LIN {X 0.002,Y -498.772,Z 962.107,A 0.000,B 0.000,C 90.000,E1 235.229} C_DIS
LIN {X -0.113,Y -494.068,Z 962.095,A 0.000,B 0.000,C 90.000,E1 233.130} C_DIS
LIN {X -0.156,Y -489.223,Z 962.083,A 0.000,B 0.000,C 90.000,E1 231.009} C_DIS
LIN {X -0.020,Y -484.237,Z 962.071,A 0.000,B 0.000,C 90.000,E1 228.852} C_DIS
LIN {X -0.074,Y -479.355,Z 962.059,A 0.000,B 0.000,C 90.000,E1 226.701} C_DIS
LIN {X -0.051,Y -475.254,Z 962.049,A 0.000,B 0.000,C 90.000,E1 224.838} C_DIS
LIN {X 0.307,Y -470.435,Z 962.037,A 0.000,B 0.000,C 90.000,E1 222.609} C_DIS
LIN {X -0.169,Y -466.298,Z 962.026,A 0.000,B 0.000,C 90.000,E1 220.782} C_DIS
LIN {X 0.117,Y -463.523,Z 962.019,A 0.000,B 0.000,C 90.000,E1 219.483} C_DIS
LIN {X -0.073,Y -458.612,Z 962.007,A 0.000,B 0.000,C 90.000,E1 217.282} C_DIS
LIN {X -0.034,Y -454.314,Z 961.996,A 0.000,B 0.000,C 90.000,E1 215.358} C_DIS
LIN {X 0.095,Y -449.373,Z 961.984,A 0.000,B 0.000,C 90.000,E1 213.086} C_DIS
LIN {X 0.228,Y -444.453,Z 961.971,A 0.000,B 0.000,C 90.000,E1 210.797} C_DIS
LIN {X -0.008,Y -439.493,Z 961.959,A 0.000,B 0.000,C 90.000,E1 208.537} C_DIS
LIN {X -0.041,Y -435.155,Z 961.948,A 0.000,B 0.000,C 90.000,E1 206.565} C_DIS
LIN {X 0.022,Y -431.464,Z 961.938,A 0.000,B 0.000,C 90.000,E1 204.899} C_DIS
LIN {X 0.016,Y -428.364,Z 961.931,A 0.000,B 0.000,C 90.000,E1 203.567} C_DIS
LIN {X -0.074,Y -421.639,Z 961.914,A 0.000,B 0.000,C 90.000,E1 200.556} C_DIS
LIN {X -0.162,Y -418.818,Z 961.907,A 0.000,B 0.000,C 90.000,E1 199.214} C_DIS
LIN {X 0.032,Y -414.002,Z 961.893,A 0.000,B 0.000,C 90.000,E1 196.804} C_DIS
LIN {X 0.082,Y -411.371,Z 961.886,A 0.000,B 0.000,C 90.000,E1 195.426} C_DIS
LIN {X -0.005,Y -407.947,Z 961.876,A 0.000,B 0.000,C 90.000,E1 193.716} C_DIS
LIN {X -0.164,Y -405.246,Z 961.869,A 0.000,B 0.000,C 90.000,E1 192.355} C_DIS
LIN {X -0.068,Y -401.253,Z 961.857,A 0.000,B 0.000,C 90.000,E1 190.254} C_DIS
LIN {X -0.122,Y -397.922,Z 961.847,A 0.000,B 0.000,C 90.000,E1 188.511} C_DIS
LIN {X -0.111,Y -392.119,Z 961.830,A 0.000,B 0.000,C 90.000,E1 185.334} C_DIS
LIN {X -0.093,Y -389.441,Z 961.820,A 0.000,B 0.000,C 90.000,E1 183.555} C_DIS
LIN {X -0.182,Y -388.975,Z 961.818,A 0.000,B 0.000,C 90.000,E1 183.212} C_DIS
LIN {X -0.048,Y -388.111,Z 961.812,A 0.000,B 0.000,C 90.000,E1 182.121} C_DIS
LIN {X 0.165,Y -387.977,Z 961.808,A 0.000,B 0.000,C 90.000,E1 181.375} C_DIS
LIN {X -0.023,Y -388.436,Z 961.804,A 0.000,B 0.000,C 90.000,E1 180.688} C_DIS
LIN {X -0.115,Y -388.908,Z 961.802,A 0.000,B 0.000,C 90.000,E1 180.344} C_DIS
LIN {X 0.138,Y -390.130,Z 961.799,A 0.000,B 0.000,C 90.000,E1 179.771} C_DIS
LIN {X 0.191,Y -391.585,Z 961.797,A 0.000,B 0.000,C 90.000,E1 179.370} C_DIS
LIN {X 0.109,Y -393.003,Z 961.795,A 0.000,B 0.000,C 90.000,E1 179.026} C_DIS
LIN {X 0.031,Y -394.990,Z 961.793,A 0.000,B 0.000,C 90.000,E1 178.682} C_DIS
LIN {X 0.104,Y -398.169,Z 961.790,A 0.000,B 0.000,C 90.000,E1 178.224} C_DIS
LIN {X -0.090,Y -402.312,Z 961.788,A 0.000,B 0.000,C 90.000,E1 177.764} C_DIS
LIN {X -0.070,Y -408.333,Z 961.784,A 0.000,B 0.000,C 90.000,E1 177.192} C_DIS
LIN {X -0.198,Y -420.662,Z 961.778,A 0.000,B 0.000,C 90.000,E1 176.102} C_DIS
LIN {X -0.071,Y -429.525,Z 961.774,A 0.000,B 0.000,C 90.000,E1 175.298} C_DIS
LIN {X -0.092,Y -438.634,Z 961.769,A 0.000,B 0.000,C 90.000,E1 174.489} C_DIS
LIN {X 0.100,Y -447.490,Z 961.765,A 0.000,B 0.000,C 90.000,E1 173.628} C_DIS
LIN {X -0.043,Y -454.687,Z 961.761,A 0.000,B 0.000,C 90.000,E1 172.932} C_DIS
LIN {X -0.092,Y -460.322,Z 961.758,A 0.000,B 0.000,C 90.000,E1 172.356} C_DIS
LIN {X 0.185,Y -468.563,Z 961.753,A 0.000,B 0.000,C 90.000,E1 171.432} C_DIS
LIN {X 0.154,Y -474.872,Z 961.749,A 0.000,B 0.000,C 90.000,E1 170.735} C_DIS
LIN {X 0.189,Y -482.568,Z 961.744,A 0.000,B 0.000,C 90.000,E1 169.803} C_DIS
LIN {X 0.051,Y -488.804,Z 961.739,A 0.000,B 0.000,C 90.000,E1 169.050} C_DIS
LIN {X 0.203,Y -495.887,Z 961.734,A 0.000,B 0.000,C 90.000,E1 168.117} C_DIS
LIN {X 0.132,Y -500.316,Z 961.731,A 0.000,B 0.000,C 90.000,E1 167.521} C_DIS
LIN {X -0.132,Y -508.811,Z 961.724,A 0.000,B 0.000,C 90.000,E1 166.353} C_DIS
LIN {X -0.165,Y -516.756,Z 961.718,A 0.000,B 0.000,C 90.000,E1 165.172} C_DIS
LIN {X -0.265,Y -523.259,Z 961.712,A 0.000,B 0.000,C 90.000,E1 164.157} C_DIS
LIN {X 0.228,Y -529.654,Z 961.706,A 0.000,B 0.000,C 90.000,E1 163.087} C_DIS
LIN {X -0.270,Y -540.981,Z 961.696,A 0.000,B 0.000,C 90.000,E1 161.275} C_DIS
LIN {X -0.336,Y -548.482,Z 961.689,A 0.000,B 0.000,C 90.000,E1 160.007} C_DIS
LIN {X 0.063,Y -552.643,Z 961.685,A 0.000,B 0.000,C 90.000,E1 159.263} C_DIS
LIN {X 0.083,Y -558.360,Z 961.679,A 0.000,B 0.000,C 90.000,E1 158.284} C_DIS
LIN {X 0.171,Y -561.441,Z 961.676,A 0.000,B 0.000,C 90.000,E1 157.720} C_DIS
LIN {X 0.199,Y -567.306,Z 961.670,A 0.000,B 0.000,C 90.000,E1 156.613} C_DIS
LIN {X 0.094,Y -572.082,Z 961.665,A 0.000,B 0.000,C 90.000,E1 155.665} C_DIS
LIN {X 0.207,Y -575.439,Z 961.661,A 0.000,B 0.000,C 90.000,E1 154.973} C_DIS
LIN {X -0.175,Y -578.579,Z 961.657,A 0.000,B 0.000,C 90.000,E1 154.332} C_DIS
LIN {X 0.174,Y -584.416,Z 961.650,A 0.000,B 0.000,C 90.000,E1 152.948} C_DIS
LIN {X 0.072,Y -587.609,Z 961.645,A 0.000,B 0.000,C 90.000,E1 152.153} C_DIS
LIN {X -0.203,Y -592.331,Z 961.638,A 0.000,B 0.000,C 90.000,E1 150.845} C_DIS
LIN {X 0.207,Y -595.985,Z 961.632,A 0.000,B 0.000,C 90.000,E1 149.744} C_DIS
LIN {X -0.231,Y -601.336,Z 961.623,A 0.000,B 0.000,C 90.000,E1 148.201} C_DIS
LIN {X -0.051,Y -608.089,Z 961.612,A 0.000,B 0.000,C 90.000,E1 146.087} C_DIS
LIN {X -0.141,Y -614.086,Z 961.602,A 0.000,B 0.000,C 90.000,E1 144.276} C_DIS
LIN {X -0.226,Y -619.902,Z 961.591,A 0.000,B 0.000,C 90.000,E1 142.477} C_DIS
LIN {X 0.032,Y -624.035,Z 961.584,A 0.000,B 0.000,C 90.000,E1 141.170} C_DIS
LIN {X 0.312,Y -631.372,Z 961.572,A 0.000,B 0.000,C 90.000,E1 138.852} C_DIS
LIN {X -0.048,Y -638.178,Z 961.560,A 0.000,B 0.000,C 90.000,E1 136.863} C_DIS
LIN {X 0.258,Y -644.183,Z 961.551,A 0.000,B 0.000,C 90.000,E1 135.081} C_DIS
LIN {X 0.159,Y -652.114,Z 961.538,A 0.000,B 0.000,C 90.000,E1 132.852} C_DIS
LIN {X 0.330,Y -660.280,Z 961.526,A 0.000,B 0.000,C 90.000,E1 130.620} C_DIS
LIN {X -0.148,Y -664.928,Z 961.519,A 0.000,B 0.000,C 90.000,E1 129.439} C_DIS
LIN {X -0.106,Y -667.632,Z 961.515,A 0.000,B 0.000,C 90.000,E1 128.705} C_DIS
LIN {X -0.048,Y -671.179,Z 961.510,A 0.000,B 0.000,C 90.000,E1 127.729} C_DIS
LIN {X 0.168,Y -675.377,Z 961.503,A 0.000,B 0.000,C 90.000,E1 126.503} C_DIS
LIN {X -0.098,Y -677.796,Z 961.499,A 0.000,B 0.000,C 90.000,E1 125.804} C_DIS
LIN {X -0.174,Y -681.560,Z 961.492,A 0.000,B 0.000,C 90.000,E1 124.612} C_DIS
LIN {X 0.184,Y -684.351,Z 961.487,A 0.000,B 0.000,C 90.000,E1 123.627} C_DIS
LIN {X -0.177,Y -687.537,Z 961.480,A 0.000,B 0.000,C 90.000,E1 122.467} C_DIS
LIN {X -0.126,Y -689.987,Z 961.475,A 0.000,B 0.000,C 90.000,E1 121.514} C_DIS
LIN {X 0.190,Y -692.197,Z 961.470,A 0.000,B 0.000,C 90.000,E1 120.541} C_DIS
LIN {X -0.292,Y -693.641,Z 961.466,A 0.000,B 0.000,C 90.000,E1 119.873} C_DIS
LIN {X -0.161,Y -694.952,Z 961.462,A 0.000,B 0.000,C 90.000,E1 119.155} C_DIS
LIN {X -0.115,Y -696.465,Z 961.455,A 0.000,B 0.000,C 90.000,E1 117.975} C_DIS
LIN {X 0.043,Y -697.251,Z 961.451,A 0.000,B 0.000,C 90.000,E1 117.257} C_DIS
LIN {X -0.206,Y -698.130,Z 961.445,A 0.000,B 0.000,C 90.000,E1 116.104} C_DIS
LIN {X 0.187,Y -698.621,Z 961.438,A 0.000,B 0.000,C 90.000,E1 114.899} C_DIS
LIN {X -0.210,Y -698.721,Z 961.436,A 0.000,B 0.000,C 90.000,E1 114.463} C_DIS
LIN {X 0.054,Y -698.680,Z 961.435,A 0.000,B 0.000,C 90.000,E1 114.207} C_DIS
LIN {X -0.340,Y -698.341,Z 961.432,A 0.000,B 0.000,C 90.000,E1 113.770} C_DIS
LIN {X 0.182,Y -697.167,Z 961.429,A 0.000,B 0.000,C 90.000,E1 113.259} C_DIS
LIN {X 0.165,Y -696.462,Z 961.428,A 0.000,B 0.000,C 90.000,E1 113.025} C_DIS
LIN {X -0.220,Y -695.014,Z 961.427,A 0.000,B 0.000,C 90.000,E1 112.823} C_DIS
LIN {X -0.117,Y -692.305,Z 961.425,A 0.000,B 0.000,C 90.000,E1 112.461} C_DIS
LIN {X 0.004,Y -691.173,Z 961.424,A 0.000,B 0.000,C 90.000,E1 112.333} C_DIS
LIN {X 0.121,Y -689.434,Z 961.423,A 0.000,B 0.000,C 90.000,E1 112.206} C_DIS
LIN {X -0.041,Y -683.525,Z 961.422,A 0.000,B 0.000,C 90.000,E1 111.950} C_DIS
LIN {X 0.173,Y -679.388,Z 961.421,A 0.000,B 0.000,C 90.000,E1 111.791} C_DIS
LIN {X -0.228,Y -677.435,Z 961.421,A 0.000,B 0.000,C 90.000,E1 111.770} C_DIS
LIN {X -0.251,Y -674.935,Z 961.421,A 0.000,B 0.000,C 90.000,E1 111.716} C_DIS
LIN {X -0.095,Y -667.646,Z 961.420,A 0.000,B 0.000,C 90.000,E1 111.663} C_DIS
LIN {X -0.128,Y -628.953,Z 961.420,A 0.000,B 0.000,C 90.000,E1 111.663} C_DIS
LIN {X 0.227,Y -623.063,Z 961.420,A 0.000,B 0.000,C 90.000,E1 111.535} C_DIS
LIN {X -0.156,Y -616.228,Z 961.419,A 0.000,B 0.000,C 90.000,E1 111.408} C_DIS
LIN {X 0.114,Y -609.362,Z 961.418,A 0.000,B 0.000,C 90.000,E1 111.153} C_DIS
LIN {X 0.021,Y -606.468,Z 961.417,A 0.000,B 0.000,C 90.000,E1 111.046} C_DIS
LIN {X -0.108,Y -599.985,Z 961.415,A 0.000,B 0.000,C 90.000,E1 110.737} C_DIS
LIN {X 0.314,Y -593.503,Z 961.413,A 0.000,B 0.000,C 90.000,E1 110.301} C_DIS
LIN {X 0.129,Y -584.030,Z 961.409,A 0.000,B 0.000,C 90.000,E1 109.631} C_DIS
LIN {X 0.293,Y -575.275,Z 961.406,A 0.000,B 0.000,C 90.000,E1 108.960} C_DIS
LIN {X -0.143,Y -567.394,Z 961.403,A 0.000,B 0.000,C 90.000,E1 108.544} C_DIS
LIN {X 0.139,Y -553.077,Z 961.399,A 0.000,B 0.000,C 90.000,E1 107.819} C_DIS
LIN {X -0.272,Y -550.970,Z 961.398,A 0.000,B 0.000,C 90.000,E1 107.638} C_DIS
LIN {X 0.213,Y -550.938,Z 961.398,A 0.000,B 0.000,C 90.000,E1 107.583} C_DIS
LIN {X -0.167,Y -550.493,Z 961.397,A 0.000,B 0.000,C 90.000,E1 107.457} C_DIS
LIN {X 0.192,Y -550.350,Z 961.394,A 0.000,B 0.000,C 90.000,E1 106.858} C_DIS
LIN {X 0.057,Y -550.977,Z 961.384,A 0.000,B 0.000,C 90.000,E1 105.190} C_DIS
LIN {X 0.153,Y -552.146,Z 961.372,A 0.000,B 0.000,C 90.000,E1 102.939} C_DIS
LIN {X -0.246,Y -554.640,Z 961.355,A 0.000,B 0.000,C 90.000,E1 99.905} C_DIS
LIN {X -0.245,Y -555.958,Z 961.347,A 0.000,B 0.000,C 90.000,E1 98.511} C_DIS
LIN {X 0.251,Y -557.272,Z 961.339,A 0.000,B 0.000,C 90.000,E1 97.068} C_DIS
LIN {X 0.149,Y -558.100,Z 961.333,A 0.000,B 0.000,C 90.000,E1 95.967} C_DIS
LIN {X 0.066,Y -559.114,Z 961.326,A 0.000,B 0.000,C 90.000,E1 94.588} C_DIS
LIN {X 0.175,Y -560.219,Z 961.315,A 0.000,B 0.000,C 90.000,E1 92.636} C_DIS
LIN {X 0.096,Y -560.910,Z 961.307,A 0.000,B 0.000,C 90.000,E1 91.260} C_DIS
LIN {X -0.080,Y -561.411,Z 961.301,A 0.000,B 0.000,C 90.000,E1 90.172} C_DIS
LIN {X -0.150,Y -561.855,Z 961.293,A 0.000,B 0.000,C 90.000,E1 88.797} C_DIS
LIN {X -0.104,Y -562.253,Z 961.284,A 0.000,B 0.000,C 90.000,E1 87.135} C_DIS
LIN {X -0.113,Y -562.489,Z 961.276,A 0.000,B 0.000,C 90.000,E1 85.755} C_DIS
LIN {X -0.026,Y -562.713,Z 961.267,A 0.000,B 0.000,C 90.000,E1 84.090} C_DIS
LIN {X 0.031,Y -562.924,Z 961.260,A 0.000,B 0.000,C 90.000,E1 82.704} C_DIS
LIN {X 0.245,Y -563.276,Z 961.250,A 0.000,B 0.000,C 90.000,E1 81.027} C_DIS
LIN {X -0.226,Y -564.154,Z 961.238,A 0.000,B 0.000,C 90.000,E1 78.870} C_DIS
LIN {X -0.171,Y -565.125,Z 961.227,A 0.000,B 0.000,C 90.000,E1 76.937} C_DIS
LIN {X -0.134,Y -566.143,Z 961.218,A 0.000,B 0.000,C 90.000,E1 75.283} C_DIS
LIN {X 0.239,Y -567.482,Z 961.208,A 0.000,B 0.000,C 90.000,E1 73.323} C_DIS
LIN {X -0.238,Y -568.369,Z 961.200,A 0.000,B 0.000,C 90.000,E1 72.000} C_DIS
LIN {X 0.172,Y -569.291,Z 961.191,A 0.000,B 0.000,C 90.000,E1 70.315} C_DIS
LIN {X -0.284,Y -570.013,Z 961.182,A 0.000,B 0.000,C 90.000,E1 68.720} C_DIS
LIN {X 0.236,Y -570.324,Z 961.177,A 0.000,B 0.000,C 90.000,E1 67.847} C_DIS
LIN {X 0.023,Y -570.847,Z 961.168,A 0.000,B 0.000,C 90.000,E1 66.230} C_DIS
LIN {X 0.219,Y -571.193,Z 961.160,A 0.000,B 0.000,C 90.000,E1 64.845} C_DIS
LIN {X -0.265,Y -571.517,Z 961.151,A 0.000,B 0.000,C 90.000,E1 63.256} C_DIS
LIN {X 0.182,Y -571.720,Z 961.144,A 0.000,B 0.000,C 90.000,E1 61.847} C_DIS
LIN {X -0.100,Y -571.827,Z 961.136,A 0.000,B 0.000,C 90.000,E1 60.511} C_DIS
LIN {X 0.080,Y -572.018,Z 961.126,A 0.000,B 0.000,C 90.000,E1 58.584} C_DIS
LIN {X -0.188,Y -572.093,Z 961.118,A 0.000,B 0.000,C 90.000,E1 57.248} C_DIS
LIN {X -0.020,Y -571.806,Z 961.109,A 0.000,B 0.000,C 90.000,E1 55.595} C_DIS
LIN {X 0.329,Y -571.460,Z 961.101,A 0.000,B 0.000,C 90.000,E1 54.196} C_DIS
LIN {X 0.073,Y -570.984,Z 961.095,A 0.000,B 0.000,C 90.000,E1 53.130} C_DIS
LIN {X 0.156,Y -570.251,Z 961.089,A 0.000,B 0.000,C 90.000,E1 52.029} C_DIS
LIN {X -0.125,Y -569.304,Z 961.083,A 0.000,B 0.000,C 90.000,E1 50.964} C_DIS
LIN {X 0.294,Y -568.235,Z 961.077,A 0.000,B 0.000,C 90.000,E1 49.828} C_DIS
LIN {X 0.215,Y -567.228,Z 961.072,A 0.000,B 0.000,C 90.000,E1 49.013} C_DIS
LIN {X -0.303,Y -566.025,Z 961.068,A 0.000,B 0.000,C 90.000,E1 48.243} C_DIS
LIN {X 0.064,Y -564.090,Z 961.062,A 0.000,B 0.000,C 90.000,E1 47.106} C_DIS
LIN {X 0.372,Y -561.923,Z 961.056,A 0.000,B 0.000,C 90.000,E1 45.972} C_DIS
LIN {X 0.189,Y -559.978,Z 961.051,A 0.000,B 0.000,C 90.000,E1 45.162} C_DIS
LIN {X -0.012,Y -557.802,Z 961.046,A 0.000,B 0.000,C 90.000,E1 44.352} C_DIS
LIN {X -0.236,Y -555.254,Z 961.042,A 0.000,B 0.000,C 90.000,E1 43.542} C_DIS
LIN {X 0.264,Y -553.483,Z 961.039,A 0.000,B 0.000,C 90.000,E1 42.933} C_DIS
LIN {X -0.028,Y -551.510,Z 961.036,A 0.000,B 0.000,C 90.000,E1 42.405} C_DIS
LIN {X 0.086,Y -548.196,Z 961.031,A 0.000,B 0.000,C 90.000,E1 41.553} C_DIS
LIN {X -0.037,Y -545.280,Z 961.027,A 0.000,B 0.000,C 90.000,E1 40.862} C_DIS
LIN {X -0.029,Y -542.661,Z 961.024,A 0.000,B 0.000,C 90.000,E1 40.297} C_DIS
LIN {X 0.021,Y -539.856,Z 961.021,A 0.000,B 0.000,C 90.000,E1 39.725} C_DIS
LIN {X -0.013,Y -533.798,Z 961.014,A 0.000,B 0.000,C 90.000,E1 38.588} C_DIS
LIN {X -0.035,Y -528.791,Z 961.010,A 0.000,B 0.000,C 90.000,E1 37.729} C_DIS
LIN {X 0.032,Y -522.690,Z 961.004,A 0.000,B 0.000,C 90.000,E1 36.710} C_DIS
LIN {X -0.234,Y -518.057,Z 961.000,A 0.000,B 0.000,C 90.000,E1 36.011} C_DIS
LIN {X -0.004,Y -512.279,Z 960.995,A 0.000,B 0.000,C 90.000,E1 35.105} C_DIS
LIN {X -0.166,Y -508.091,Z 960.992,A 0.000,B 0.000,C 90.000,E1 34.532} C_DIS
LIN {X 0.057,Y -503.632,Z 960.988,A 0.000,B 0.000,C 90.000,E1 33.913} C_DIS
LIN {X 0.244,Y -498.877,Z 960.985,A 0.000,B 0.000,C 90.000,E1 33.293} C_DIS
LIN {X -0.086,Y -495.051,Z 960.983,A 0.000,B 0.000,C 90.000,E1 32.880} C_DIS
LIN {X 0.081,Y -488.398,Z 960.979,A 0.000,B 0.000,C 90.000,E1 32.133} C_DIS
LIN {X 0.073,Y -481.531,Z 960.975,A 0.000,B 0.000,C 90.000,E1 31.416} C_DIS
LIN {X -0.107,Y -471.350,Z 960.969,A 0.000,B 0.000,C 90.000,E1 30.463} C_DIS
LIN {X 0.183,Y -463.949,Z 960.965,A 0.000,B 0.000,C 90.000,E1 29.745} C_DIS
LIN {X 0.171,Y -455.058,Z 960.961,A 0.000,B 0.000,C 90.000,E1 28.949} C_DIS
LIN {X 0.248,Y -442.802,Z 960.955,A 0.000,B 0.000,C 90.000,E1 27.897} C_DIS
LIN {X -0.116,Y -423.164,Z 960.946,A 0.000,B 0.000,C 90.000,E1 26.232} C_DIS
LIN {X 0.066,Y -406.759,Z 960.937,A 0.000,B 0.000,C 90.000,E1 24.643} C_DIS
LIN {X 0.050,Y -398.631,Z 960.932,A 0.000,B 0.000,C 90.000,E1 23.770} C_DIS
LIN {X 0.158,Y -393.390,Z 960.928,A 0.000,B 0.000,C 90.000,E1 23.078} C_DIS
LIN {X 0.117,Y -391.309,Z 960.926,A 0.000,B 0.000,C 90.000,E1 22.642} C_DIS
LIN {X 0.065,Y -390.232,Z 960.923,A 0.000,B 0.000,C 90.000,E1 22.206} C_DIS
LIN {X 0.084,Y -389.878,Z 960.922,A 0.000,B 0.000,C 90.000,E1 22.025} C_DIS
LIN {X 0.049,Y -389.531,Z 960.919,A 0.000,B 0.000,C 90.000,E1 21.408} C_DIS
LIN {X -0.156,Y -389.967,Z 960.913,A 0.000,B 0.000,C 90.000,E1 20.301} C_DIS
LIN {X 0.152,Y -392.234,Z 960.899,A 0.000,B 0.000,C 90.000,E1 17.764} C_DIS
LIN {X -0.017,Y -395.491,Z 960.883,A 0.000,B 0.000,C 90.000,E1 14.954} C_DIS
LIN {X 0.092,Y -399.231,Z 960.867,A 0.000,B 0.000,C 90.000,E1 12.119} C_DIS
LIN {X 0.072,Y -403.658,Z 960.852,A 0.000,B 0.000,C 90.000,E1 9.321} C_DIS
LIN {X 0.020,Y -408.661,Z 960.836,A 0.000,B 0.000,C 90.000,E1 6.549} C_DIS
LIN {X 0.118,Y -415.635,Z 960.817,A 0.000,B 0.000,C 90.000,E1 3.094} C_DIS
LIN {X -0.144,Y -420.986,Z 960.804,A 0.000,B 0.000,C 90.000,E1 0.745} C_DIS
LIN {X 0.000,Y -422.737,Z 960.800,A 0.000,B 0.000,C 90.000,E1 360.000} C_DIS
LIN {X -0.053,Y -425.183,Z 960.796,A 0.000,B 0.000,C 90.000,E1 359.312} C_DIS
LIN {X -0.118,Y -428.115,Z 960.793,A 0.000,B 0.000,C 90.000,E1 358.797} C_DIS
LIN {X 0.142,Y -429.485,Z 960.792,A 0.000,B 0.000,C 90.000,E1 358.511} C_DIS
LIN {X -0.025,Y -432.070,Z 960.790,A 0.000,B 0.000,C 90.000,E1 358.282} C_DIS
LIN {X 0.079,Y -434.973,Z 960.789,A 0.000,B 0.000,C 90.000,E1 357.993} C_DIS
LIN {X -0.159,Y -441.329,Z 960.787,A 0.000,B 0.000,C 90.000,E1 357.650} C_DIS
LIN {X -0.090,Y -450.033,Z 960.784,A 0.000,B 0.000,C 90.000,E1 357.192} C_DIS
LIN {X -0.185,Y -465.315,Z 960.780,A 0.000,B 0.000,C 90.000,E1 356.388} C_DIS
LIN {X -0.060,Y -473.709,Z 960.777,A 0.000,B 0.000,C 90.000,E1 355.927} C_DIS
LIN {X 0.093,Y -483.670,Z 960.774,A 0.000,B 0.000,C 90.000,E1 355.355} C_DIS
LIN {X -0.153,Y -493.694,Z 960.771,A 0.000,B 0.000,C 90.000,E1 354.837} C_DIS
LIN {X -0.022,Y -503.392,Z 960.768,A 0.000,B 0.000,C 90.000,E1 354.261} C_DIS
LIN {X -0.111,Y -512.933,Z 960.765,A 0.000,B 0.000,C 90.000,E1 353.685} C_DIS
LIN {X 0.191,Y -523.897,Z 960.761,A 0.000,B 0.000,C 90.000,E1 352.932} C_DIS
LIN {X -0.019,Y -531.408,Z 960.758,A 0.000,B 0.000,C 90.000,E1 352.413} C_DIS
LIN {X 0.158,Y -539.663,Z 960.754,A 0.000,B 0.000,C 90.000,E1 351.724} C_DIS
LIN {X -0.121,Y -546.547,Z 960.751,A 0.000,B 0.000,C 90.000,E1 351.141} C_DIS
LIN {X 0.086,Y -550.532,Z 960.749,A 0.000,B 0.000,C 90.000,E1 350.735} C_DIS
LIN {X 0.116,Y -556.731,Z 960.745,A 0.000,B 0.000,C 90.000,E1 350.095} C_DIS
LIN {X 0.204,Y -562.520,Z 960.741,A 0.000,B 0.000,C 90.000,E1 349.398} C_DIS
LIN {X -0.033,Y -566.889,Z 960.738,A 0.000,B 0.000,C 90.000,E1 348.870} C_DIS
LIN {X -0.051,Y -572.834,Z 960.734,A 0.000,B 0.000,C 90.000,E1 348.049} C_DIS
LIN {X -0.007,Y -578.239,Z 960.729,A 0.000,B 0.000,C 90.000,E1 347.229} C_DIS
LIN {X -0.243,Y -584.758,Z 960.723,A 0.000,B 0.000,C 90.000,E1 346.172} C_DIS
LIN {X 0.319,Y -590.677,Z 960.717,A 0.000,B 0.000,C 90.000,E1 345.046} C_DIS
LIN {X 0.197,Y -594.182,Z 960.713,A 0.000,B 0.000,C 90.000,E1 344.393} C_DIS
LIN {X -0.193,Y -598.774,Z 960.708,A 0.000,B 0.000,C 90.000,E1 343.504} C_DIS
LIN {X -0.308,Y -602.563,Z 960.704,A 0.000,B 0.000,C 90.000,E1 342.725} C_DIS
LIN {X 0.102,Y -607.289,Z 960.698,A 0.000,B 0.000,C 90.000,E1 341.638} C_DIS
LIN {X 0.003,Y -611.744,Z 960.692,A 0.000,B 0.000,C 90.000,E1 340.604} C_DIS
LIN {X -0.038,Y -615.949,Z 960.687,A 0.000,B 0.000,C 90.000,E1 339.571} C_DIS
LIN {X -0.028,Y -619.866,Z 960.681,A 0.000,B 0.000,C 90.000,E1 338.539} C_DIS
LIN {X -0.309,Y -622.627,Z 960.677,A 0.000,B 0.000,C 90.000,E1 337.794} C_DIS
LIN {X 0.016,Y -626.085,Z 960.671,A 0.000,B 0.000,C 90.000,E1 336.741} C_DIS
LIN {X -0.190,Y -629.362,Z 960.665,A 0.000,B 0.000,C 90.000,E1 335.741} C_DIS
LIN {X -0.088,Y -632.438,Z 960.660,A 0.000,B 0.000,C 90.000,E1 334.717} C_DIS
LIN {X 0.023,Y -634.596,Z 960.655,A 0.000,B 0.000,C 90.000,E1 333.948} C_DIS
LIN {X -0.083,Y -637.250,Z 960.650,A 0.000,B 0.000,C 90.000,E1 332.948} C_DIS
LIN {X -0.140,Y -639.713,Z 960.644,A 0.000,B 0.000,C 90.000,E1 331.948} C_DIS
LIN {X -0.326,Y -643.097,Z 960.636,A 0.000,B 0.000,C 90.000,E1 330.461} C_DIS
LIN {X -0.215,Y -645.673,Z 960.629,A 0.000,B 0.000,C 90.000,E1 329.203} C_DIS
LIN {X -0.143,Y -647.422,Z 960.623,A 0.000,B 0.000,C 90.000,E1 328.201} C_DIS
LIN {X -0.053,Y -649.027,Z 960.618,A 0.000,B 0.000,C 90.000,E1 327.199} C_DIS
LIN {X -0.134,Y -650.356,Z 960.612,A 0.000,B 0.000,C 90.000,E1 326.215} C_DIS
LIN {X -0.115,Y -651.840,Z 960.605,A 0.000,B 0.000,C 90.000,E1 324.975} C_DIS
LIN {X 0.300,Y -653.096,Z 960.599,A 0.000,B 0.000,C 90.000,E1 323.703} C_DIS
LIN {X -0.174,Y -653.690,Z 960.594,A 0.000,B 0.000,C 90.000,E1 323.004} C_DIS
LIN {X 0.205,Y -654.407,Z 960.589,A 0.000,B 0.000,C 90.000,E1 321.984} C_DIS
LIN {X 0.029,Y -655.594,Z 960.579,A 0.000,B 0.000,C 90.000,E1 320.275} C_DIS
LIN {X -0.070,Y -656.084,Z 960.574,A 0.000,B 0.000,C 90.000,E1 319.299} C_DIS
LIN {X 0.182,Y -657.205,Z 960.563,A 0.000,B 0.000,C 90.000,E1 317.310} C_DIS
LIN {X 0.025,Y -658.395,Z 960.555,A 0.000,B 0.000,C 90.000,E1 315.850} C_DIS
LIN {X 0.360,Y -659.412,Z 960.548,A 0.000,B 0.000,C 90.000,E1 314.595} C_DIS
LIN {X -0.287,Y -661.344,Z 960.536,A 0.000,B 0.000,C 90.000,E1 312.447} C_DIS
LIN {X -0.335,Y -662.436,Z 960.529,A 0.000,B 0.000,C 90.000,E1 311.229} C_DIS
LIN {X -0.364,Y -663.381,Z 960.522,A 0.000,B 0.000,C 90.000,E1 310.011} C_DIS
LIN {X 0.126,Y -664.202,Z 960.515,A 0.000,B 0.000,C 90.000,E1 308.749} C_DIS
LIN {X 0.218,Y -664.932,Z 960.509,A 0.000,B 0.000,C 90.000,E1 307.523} C_DIS
LIN {X 0.323,Y -665.435,Z 960.502,A 0.000,B 0.000,C 90.000,E1 306.297} C_DIS
LIN {X -0.076,Y -665.738,Z 960.496,A 0.000,B 0.000,C 90.000,E1 305.358} C_DIS
LIN {X -0.036,Y -666.325,Z 960.484,A 0.000,B 0.000,C 90.000,E1 303.166} C_DIS
LIN {X -0.320,Y -667.428,Z 960.472,A 0.000,B 0.000,C 90.000,E1 301.003} C_DIS
LIN {X -0.277,Y -670.510,Z 960.455,A 0.000,B 0.000,C 90.000,E1 297.847} C_DIS
LIN {X -0.050,Y -674.365,Z 960.441,A 0.000,B 0.000,C 90.000,E1 295.412} C_DIS
LIN {X -0.038,Y -676.555,Z 960.435,A 0.000,B 0.000,C 90.000,E1 294.207} C_DIS
LIN {X -0.189,Y -678.094,Z 960.429,A 0.000,B 0.000,C 90.000,E1 293.259} C_DIS
LIN {X -0.080,Y -678.727,Z 960.427,A 0.000,B 0.000,C 90.000,E1 292.770} C_DIS
LIN {X 0.038,Y -678.858,Z 960.424,A 0.000,B 0.000,C 90.000,E1 292.280} C_DIS
LIN {X 0.226,Y -678.825,Z 960.423,A 0.000,B 0.000,C 90.000,E1 292.025} C_DIS
LIN {X -0.284,Y -678.126,Z 960.420,A 0.000,B 0.000,C 90.000,E1 291.589} C_DIS
LIN {X -0.102,Y -677.484,Z 960.419,A 0.000,B 0.000,C 90.000,E1 291.334} C_DIS
LIN {X -0.257,Y -676.818,Z 960.418,A 0.000,B 0.000,C 90.000,E1 291.227} C_DIS
LIN {X 0.007,Y -674.111,Z 960.416,A 0.000,B 0.000,C 90.000,E1 290.844} C_DIS
LIN {X -0.148,Y -673.175,Z 960.415,A 0.000,B 0.000,C 90.000,E1 290.737} C_DIS
LIN {X -0.064,Y -672.011,Z 960.414,A 0.000,B 0.000,C 90.000,E1 290.610} C_DIS
LIN {X 0.094,Y -668.492,Z 960.413,A 0.000,B 0.000,C 90.000,E1 290.355} C_DIS
LIN {X -0.008,Y -665.690,Z 960.412,A 0.000,B 0.000,C 90.000,E1 290.174} C_DIS
LIN {X -0.357,Y -658.708,Z 960.410,A 0.000,B 0.000,C 90.000,E1 289.758} C_DIS
LIN {X -0.172,Y -657.487,Z 960.409,A 0.000,B 0.000,C 90.000,E1 289.631} C_DIS
LIN {X -0.213,Y -657.465,Z 960.409,A 0.000,B 0.000,C 90.000,E1 289.631} C_DIS
LIN {X 0.130,Y -657.090,Z 960.408,A 0.000,B 0.000,C 90.000,E1 289.450} C_DIS
LIN {X 0.187,Y -657.585,Z 960.406,A 0.000,B 0.000,C 90.000,E1 289.141} C_DIS
LIN {X 0.068,Y -658.610,Z 960.405,A 0.000,B 0.000,C 90.000,E1 288.906} C_DIS
LIN {X 0.002,Y -660.361,Z 960.403,A 0.000,B 0.000,C 90.000,E1 288.544} C_DIS
LIN {X -0.048,Y -665.331,Z 960.398,A 0.000,B 0.000,C 90.000,E1 287.692} C_DIS
LIN {X -0.225,Y -668.047,Z 960.396,A 0.000,B 0.000,C 90.000,E1 287.221} C_DIS
LIN {X -0.188,Y -670.450,Z 960.393,A 0.000,B 0.000,C 90.000,E1 286.732} C_DIS
LIN {X 0.251,Y -673.571,Z 960.389,A 0.000,B 0.000,C 90.000,E1 285.969} C_DIS
LIN {X 0.259,Y -675.833,Z 960.385,A 0.000,B 0.000,C 90.000,E1 285.245} C_DIS
LIN {X 0.157,Y -677.084,Z 960.382,A 0.000,B 0.000,C 90.000,E1 284.773} C_DIS
LIN {X 0.018,Y -678.602,Z 960.378,A 0.000,B 0.000,C 90.000,E1 284.064} C_DIS
LIN {X -0.145,Y -680.106,Z 960.373,A 0.000,B 0.000,C 90.000,E1 283.119} C_DIS
LIN {X -0.258,Y -680.885,Z 960.369,A 0.000,B 0.000,C 90.000,E1 282.411} C_DIS
LIN {X 0.193,Y -681.244,Z 960.366,A 0.000,B 0.000,C 90.000,E1 281.895} C_DIS
LIN {X 0.088,Y -681.336,Z 960.362,A 0.000,B 0.000,C 90.000,E1 281.186} C_DIS
LIN {X 0.015,Y -681.112,Z 960.360,A 0.000,B 0.000,C 90.000,E1 280.715} C_DIS
LIN {X -0.188,Y -680.685,Z 960.357,A 0.000,B 0.000,C 90.000,E1 280.254} C_DIS
LIN {X -0.271,Y -679.901,Z 960.354,A 0.000,B 0.000,C 90.000,E1 279.782} C_DIS
LIN {X 0.195,Y -678.840,Z 960.352,A 0.000,B 0.000,C 90.000,E1 279.265} C_DIS
LIN {X 0.146,Y -678.234,Z 960.350,A 0.000,B 0.000,C 90.000,E1 279.029} C_DIS
LIN {X -0.065,Y -676.690,Z 960.348,A 0.000,B 0.000,C 90.000,E1 278.568} C_DIS
LIN {X -0.282,Y -674.910,Z 960.345,A 0.000,B 0.000,C 90.000,E1 278.106} C_DIS
LIN {X 0.160,Y -672.860,Z 960.342,A 0.000,B 0.000,C 90.000,E1 277.587} C_DIS
LIN {X -0.079,Y -669.818,Z 960.339,A 0.000,B 0.000,C 90.000,E1 277.004} C_DIS
LIN {X 0.235,Y -666.403,Z 960.336,A 0.000,B 0.000,C 90.000,E1 276.372} C_DIS
LIN {X -0.140,Y -662.282,Z 960.332,A 0.000,B 0.000,C 90.000,E1 275.796} C_DIS
LIN {X 0.208,Y -658.663,Z 960.329,A 0.000,B 0.000,C 90.000,E1 275.277} C_DIS
LIN {X -0.181,Y -654.566,Z 960.327,A 0.000,B 0.000,C 90.000,E1 274.821} C_DIS
LIN {X 0.010,Y -648.911,Z 960.323,A 0.000,B 0.000,C 90.000,E1 274.188} C_DIS
LIN {X 0.191,Y -642.807,Z 960.320,A 0.000,B 0.000,C 90.000,E1 273.555} C_DIS
LIN {X -0.051,Y -637.693,Z 960.317,A 0.000,B 0.000,C 90.000,E1 273.094} C_DIS
LIN {X -0.095,Y -630.897,Z 960.314,A 0.000,B 0.000,C 90.000,E1 272.522} C_DIS
LIN {X 0.122,Y -625.237,Z 960.312,A 0.000,B 0.000,C 90.000,E1 272.064} C_DIS
LIN {X 0.086,Y -617.688,Z 960.309,A 0.000,B 0.000,C 90.000,E1 271.547} C_DIS
LIN {X 0.221,Y -611.539,Z 960.307,A 0.000,B 0.000,C 90.000,E1 271.146} C_DIS
LIN {X -0.208,Y -603.442,Z 960.304,A 0.000,B 0.000,C 90.000,E1 270.745} C_DIS
LIN {X -0.006,Y -596.623,Z 960.302,A 0.000,B 0.000,C 90.000,E1 270.401} C_DIS
LIN {X 0.064,Y -591.566,Z 960.301,A 0.000,B 0.000,C 90.000,E1 270.172} C_DIS
LIN {X 0.279,Y -584.374,Z 960.300,A 0.000,B 0.000,C 90.000,E1 269.885} C_DIS
LIN {X 0.273,Y -576.976,Z 960.298,A 0.000,B 0.000,C 90.000,E1 269.656} C_DIS
LIN {X -0.115,Y -571.323,Z 960.297,A 0.000,B 0.000,C 90.000,E1 269.542} C_DIS
LIN {X -0.261,Y -564.391,Z 960.297,A 0.000,B 0.000,C 90.000,E1 269.427} C_DIS
LIN {X 0.030,Y -557.880,Z 960.296,A 0.000,B 0.000,C 90.000,E1 269.312} C_DIS
LIN {X -0.206,Y -551.016,Z 960.296,A 0.000,B 0.000,C 90.000,E1 269.312} C_DIS
LIN {X -0.139,Y -545.355,Z 960.296,A 0.000,B 0.000,C 90.000,E1 269.255} C_DIS
LIN {X -0.139,Y -543.658,Z 960.295,A 0.000,B 0.000,C 90.000,E1 269.141} C_DIS
LIN {X -0.171,Y -543.615,Z 960.295,A 0.000,B 0.000,C 90.000,E1 269.141} C_DIS
LIN {X -0.121,Y -543.318,Z 960.295,A 0.000,B 0.000,C 90.000,E1 269.026} C_DIS
LIN {X -0.139,Y -542.478,Z 960.291,A 0.000,B 0.000,C 90.000,E1 268.339} C_DIS
LIN {X 0.076,Y -540.931,Z 960.280,A 0.000,B 0.000,C 90.000,E1 266.331} C_DIS
LIN {X -0.240,Y -539.555,Z 960.269,A 0.000,B 0.000,C 90.000,E1 264.375} C_DIS
LIN {X -0.060,Y -538.288,Z 960.259,A 0.000,B 0.000,C 90.000,E1 262.648} C_DIS
LIN {X 0.109,Y -537.311,Z 960.253,A 0.000,B 0.000,C 90.000,E1 261.489} C_DIS
LIN {X -0.205,Y -535.832,Z 960.245,A 0.000,B 0.000,C 90.000,E1 260.095} C_DIS
LIN {X -0.032,Y -534.829,Z 960.240,A 0.000,B 0.000,C 90.000,E1 259.218} C_DIS
LIN {X -0.193,Y -532.360,Z 960.229,A 0.000,B 0.000,C 90.000,E1 257.229} C_DIS
LIN {X -0.273,Y -529.585,Z 960.216,A 0.000,B 0.000,C 90.000,E1 254.936} C_DIS
LIN {X 0.134,Y -528.005,Z 960.208,A 0.000,B 0.000,C 90.000,E1 253.449} C_DIS
LIN {X 0.160,Y -526.351,Z 960.200,A 0.000,B 0.000,C 90.000,E1 252.000} C_DIS
LIN {X -0.168,Y -524.147,Z 960.190,A 0.000,B 0.000,C 90.000,E1 250.296} C_DIS
LIN {X -0.186,Y -522.695,Z 960.184,A 0.000,B 0.000,C 90.000,E1 249.135} C_DIS
LIN {X 0.075,Y -520.436,Z 960.174,A 0.000,B 0.000,C 90.000,E1 247.358} C_DIS
LIN {X -0.147,Y -518.252,Z 960.166,A 0.000,B 0.000,C 90.000,E1 245.921} C_DIS
LIN {X -0.190,Y -516.026,Z 960.158,A 0.000,B 0.000,C 90.000,E1 244.460} C_DIS
LIN {X 0.074,Y -513.273,Z 960.148,A 0.000,B 0.000,C 90.000,E1 242.666} C_DIS
LIN {X 0.168,Y -510.859,Z 960.140,A 0.000,B 0.000,C 90.000,E1 241.179} C_DIS
LIN {X 0.127,Y -508.844,Z 960.133,A 0.000,B 0.000,C 90.000,E1 239.999} C_DIS
LIN {X -0.015,Y -507.166,Z 960.129,A 0.000,B 0.000,C 90.000,E1 239.125} C_DIS
LIN {X 0.147,Y -504.793,Z 960.122,A 0.000,B 0.000,C 90.000,E1 237.916} C_DIS
LIN {X -0.153,Y -502.264,Z 960.115,A 0.000,B 0.000,C 90.000,E1 236.755} C_DIS
LIN {X -0.204,Y -498.838,Z 960.107,A 0.000,B 0.000,C 90.000,E1 235.261} C_DIS
LIN {X -0.032,Y -494.135,Z 960.095,A 0.000,B 0.000,C 90.000,E1 233.130} C_DIS
LIN {X -0.074,Y -489.307,Z 960.083,A 0.000,B 0.000,C 90.000,E1 231.009} C_DIS
LIN {X 0.062,Y -484.308,Z 960.071,A 0.000,B 0.000,C 90.000,E1 228.852} C_DIS
LIN {X 0.214,Y -480.146,Z 960.061,A 0.000,B 0.000,C 90.000,E1 226.986} C_DIS
LIN {X 0.034,Y -475.327,Z 960.049,A 0.000,B 0.000,C 90.000,E1 224.838} C_DIS
LIN {X -0.271,Y -470.516,Z 960.037,A 0.000,B 0.000,C 90.000,E1 222.690} C_DIS
LIN {X -0.081,Y -466.418,Z 960.027,A 0.000,B 0.000,C 90.000,E1 220.782} C_DIS
LIN {X -0.041,Y -462.881,Z 960.018,A 0.000,B 0.000,C 90.000,E1 219.197} C_DIS
LIN {X 0.124,Y -457.986,Z 960.005,A 0.000,B 0.000,C 90.000,E1 216.950} C_DIS
LIN {X -0.204,Y -454.430,Z 959.997,A 0.000,B 0.000,C 90.000,E1 215.391} C_DIS
LIN {X 0.189,Y -449.496,Z 959.984,A 0.000,B 0.000,C 90.000,E1 213.086} C_DIS
LIN {X -0.058,Y -444.529,Z 959.971,A 0.000,B 0.000,C 90.000,E1 210.846} C_DIS
LIN {X -0.120,Y -439.600,Z 959.959,A 0.000,B 0.000,C 90.000,E1 208.565} C_DIS
LIN {X 0.058,Y -435.231,Z 959.948,A 0.000,B 0.000,C 90.000,E1 206.565} C_DIS
LIN {X 0.121,Y -431.579,Z 959.938,A 0.000,B 0.000,C 90.000,E1 204.899} C_DIS
LIN {X -0.055,Y -428.484,Z 959.931,A 0.000,B 0.000,C 90.000,E1 203.590} C_DIS
LIN {X -0.153,Y -422.456,Z 959.916,A 0.000,B 0.000,C 90.000,E1 200.918} C_DIS
LIN {X -0.230,Y -419.654,Z 959.909,A 0.000,B 0.000,C 90.000,E1 199.577} C_DIS
LIN {X 0.138,Y -414.101,Z 959.893,A 0.000,B 0.000,C 90.000,E1 196.804} C_DIS
LIN {X 0.189,Y -411.453,Z 959.886,A 0.000,B 0.000,C 90.000,E1 195.426} C_DIS
LIN {X -0.182,Y -407.353,Z 959.874,A 0.000,B 0.000,C 90.000,E1 193.411} C_DIS
LIN {X 0.043,Y -403.311,Z 959.863,A 0.000,B 0.000,C 90.000,E1 191.299} C_DIS
LIN {X 0.027,Y -400.013,Z 959.853,A 0.000,B 0.000,C 90.000,E1 189.557} C_DIS
LIN {X -0.054,Y -396.641,Z 959.843,A 0.000,B 0.000,C 90.000,E1 187.814} C_DIS
LIN {X -0.001,Y -392.133,Z 959.830,A 0.000,B 0.000,C 90.000,E1 185.334} C_DIS
LIN {X -0.074,Y -388.879,Z 959.818,A 0.000,B 0.000,C 90.000,E1 183.212} C_DIS
LIN {X 0.060,Y -387.854,Z 959.812,A 0.000,B 0.000,C 90.000,E1 182.121} C_DIS
LIN {X -0.117,Y -387.581,Z 959.808,A 0.000,B 0.000,C 90.000,E1 181.432} C_DIS
LIN {X 0.038,Y -387.839,Z 959.804,A 0.000,B 0.000,C 90.000,E1 180.630} C_DIS
LIN {X -0.149,Y -388.718,Z 959.800,A 0.000,B 0.000,C 90.000,E1 179.943} C_DIS
LIN {X 0.102,Y -389.948,Z 959.797,A 0.000,B 0.000,C 90.000,E1 179.370} C_DIS
LIN {X -0.071,Y -392.830,Z 959.793,A 0.000,B 0.000,C 90.000,E1 178.682} C_DIS
LIN {X 0.024,Y -394.378,Z 959.791,A 0.000,B 0.000,C 90.000,E1 178.396} C_DIS
LIN {X -0.120,Y -397.913,Z 959.789,A 0.000,B 0.000,C 90.000,E1 177.936} C_DIS
LIN {X -0.150,Y -400.817,Z 959.787,A 0.000,B 0.000,C 90.000,E1 177.593} C_DIS
LIN {X 0.088,Y -408.295,Z 959.783,A 0.000,B 0.000,C 90.000,E1 176.846} C_DIS
LIN {X -0.099,Y -425.468,Z 959.774,A 0.000,B 0.000,C 90.000,E1 175.355} C_DIS
LIN {X -0.010,Y -437.697,Z 959.768,A 0.000,B 0.000,C 90.000,E1 174.261} C_DIS
LIN {X -0.148,Y -446.549,Z 959.764,A 0.000,B 0.000,C 90.000,E1 173.451} C_DIS
LIN {X -0.114,Y -455.149,Z 959.759,A 0.000,B 0.000,C 90.000,E1 172.591} C_DIS
LIN {X -0.079,Y -460.804,Z 959.756,A 0.000,B 0.000,C 90.000,E1 172.008} C_DIS
LIN {X 0.079,Y -467.630,Z 959.752,A 0.000,B 0.000,C 90.000,E1 171.254} C_DIS
LIN {X 0.044,Y -474.489,Z 959.747,A 0.000,B 0.000,C 90.000,E1 170.500} C_DIS
LIN {X -0.213,Y -483.486,Z 959.741,A 0.000,B 0.000,C 90.000,E1 169.454} C_DIS
LIN {X 0.227,Y -489.734,Z 959.737,A 0.000,B 0.000,C 90.000,E1 168.634} C_DIS
LIN {X 0.008,Y -494.455,Z 959.734,A 0.000,B 0.000,C 90.000,E1 168.049} C_DIS
LIN {X 0.225,Y -501.092,Z 959.729,A 0.000,B 0.000,C 90.000,E1 167.117} C_DIS
LIN {X 0.141,Y -507.475,Z 959.724,A 0.000,B 0.000,C 90.000,E1 166.228} C_DIS
LIN {X -0.200,Y -514.592,Z 959.718,A 0.000,B 0.000,C 90.000,E1 165.227} C_DIS
LIN {X -0.009,Y -522.164,Z 959.711,A 0.000,B 0.000,C 90.000,E1 164.031} C_DIS
LIN {X -0.016,Y -530.318,Z 959.704,A 0.000,B 0.000,C 90.000,E1 162.725} C_DIS
LIN {X 0.155,Y -540.746,Z 959.695,A 0.000,B 0.000,C 90.000,E1 160.986} C_DIS
LIN {X -0.245,Y -548.358,Z 959.687,A 0.000,B 0.000,C 90.000,E1 159.752} C_DIS
LIN {X 0.002,Y -555.790,Z 959.680,A 0.000,B 0.000,C 90.000,E1 158.465} C_DIS
LIN {X 0.163,Y -560.474,Z 959.676,A 0.000,B 0.000,C 90.000,E1 157.614} C_DIS
LIN {X -0.125,Y -566.458,Z 959.670,A 0.000,B 0.000,C 90.000,E1 156.538} C_DIS
LIN {X -0.151,Y -570.602,Z 959.665,A 0.000,B 0.000,C 90.000,E1 155.717} C_DIS
LIN {X 0.310,Y -575.326,Z 959.660,A 0.000,B 0.000,C 90.000,E1 154.717} C_DIS
LIN {X 0.154,Y -576.640,Z 959.658,A 0.000,B 0.000,C 90.000,E1 154.460} C_DIS
LIN {X -0.183,Y -583.668,Z 959.649,A 0.000,B 0.000,C 90.000,E1 152.871} C_DIS
LIN {X 0.228,Y -586.858,Z 959.645,A 0.000,B 0.000,C 90.000,E1 152.025} C_DIS
LIN {X -0.058,Y -591.742,Z 959.637,A 0.000,B 0.000,C 90.000,E1 150.717} C_DIS
LIN {X -0.075,Y -594.511,Z 959.633,A 0.000,B 0.000,C 90.000,E1 149.921} C_DIS
LIN {X -0.021,Y -599.909,Z 959.624,A 0.000,B 0.000,C 90.000,E1 148.329} C_DIS
LIN {X -0.132,Y -605.861,Z 959.614,A 0.000,B 0.000,C 90.000,E1 146.501} C_DIS
LIN {X 0.016,Y -610.155,Z 959.607,A 0.000,B 0.000,C 90.000,E1 145.182} C_DIS
LIN {X 0.304,Y -613.654,Z 959.601,A 0.000,B 0.000,C 90.000,E1 144.116} C_DIS
LIN {X -0.158,Y -619.506,Z 959.591,A 0.000,B 0.000,C 90.000,E1 142.351} C_DIS
LIN {X 0.088,Y -623.654,Z 959.584,A 0.000,B 0.000,C 90.000,E1 141.045} C_DIS
LIN {X -0.220,Y -628.555,Z 959.575,A 0.000,B 0.000,C 90.000,E1 139.542} C_DIS
LIN {X 0.105,Y -632.775,Z 959.568,A 0.000,B 0.000,C 90.000,E1 138.243} C_DIS
LIN {X -0.062,Y -638.003,Z 959.560,A 0.000,B 0.000,C 90.000,E1 136.743} C_DIS
LIN {X -0.042,Y -642.348,Z 959.553,A 0.000,B 0.000,C 90.000,E1 135.486} C_DIS
LIN {X 0.432,Y -647.609,Z 959.544,A 0.000,B 0.000,C 90.000,E1 133.947} C_DIS
LIN {X -0.306,Y -652.121,Z 959.538,A 0.000,B 0.000,C 90.000,E1 132.771} C_DIS
LIN {X -0.108,Y -659.399,Z 959.527,A 0.000,B 0.000,C 90.000,E1 130.782} C_DIS
LIN {X -0.177,Y -664.057,Z 959.520,A 0.000,B 0.000,C 90.000,E1 129.564} C_DIS
LIN {X -0.093,Y -669.482,Z 959.512,A 0.000,B 0.000,C 90.000,E1 128.096} C_DIS
LIN {X 0.106,Y -672.924,Z 959.506,A 0.000,B 0.000,C 90.000,E1 127.111} C_DIS
LIN {X -0.188,Y -677.092,Z 959.500,A 0.000,B 0.000,C 90.000,E1 125.931} C_DIS
LIN {X 0.279,Y -680.885,Z 959.493,A 0.000,B 0.000,C 90.000,E1 124.692} C_DIS
LIN {X -0.314,Y -683.776,Z 959.488,A 0.000,B 0.000,C 90.000,E1 123.785} C_DIS
LIN {X 0.270,Y -686.977,Z 959.481,A 0.000,B 0.000,C 90.000,E1 122.546} C_DIS
LIN {X 0.318,Y -689.454,Z 959.476,A 0.000,B 0.000,C 90.000,E1 121.592} C_DIS
LIN {X 0.038,Y -691.703,Z 959.470,A 0.000,B 0.000,C 90.000,E1 120.669} C_DIS
LIN {X -0.210,Y -693.605,Z 959.465,A 0.000,B 0.000,C 90.000,E1 119.745} C_DIS
LIN {X -0.325,Y -694.489,Z 959.463,A 0.000,B 0.000,C 90.000,E1 119.283} C_DIS
LIN {X -0.288,Y -696.080,Z 959.456,A 0.000,B 0.000,C 90.000,E1 118.103} C_DIS
LIN {X -0.134,Y -696.878,Z 959.452,A 0.000,B 0.000,C 90.000,E1 117.385} C_DIS
LIN {X -0.389,Y -697.751,Z 959.446,A 0.000,B 0.000,C 90.000,E1 116.232} C_DIS
LIN {X -0.002,Y -698.249,Z 959.439,A 0.000,B 0.000,C 90.000,E1 115.027} C_DIS
LIN {X -0.137,Y -698.417,Z 959.435,A 0.000,B 0.000,C 90.000,E1 114.335} C_DIS
LIN {X 0.388,Y -698.116,Z 959.433,A 0.000,B 0.000,C 90.000,E1 113.823} C_DIS
LIN {X -0.271,Y -697.780,Z 959.431,A 0.000,B 0.000,C 90.000,E1 113.643} C_DIS
LIN {X -0.028,Y -696.508,Z 959.429,A 0.000,B 0.000,C 90.000,E1 113.153} C_DIS
LIN {X 0.228,Y -695.369,Z 959.427,A 0.000,B 0.000,C 90.000,E1 112.898} C_DIS
LIN {X -0.306,Y -692.954,Z 959.425,A 0.000,B 0.000,C 90.000,E1 112.589} C_DIS
LIN {X -0.183,Y -692.041,Z 959.425,A 0.000,B 0.000,C 90.000,E1 112.461} C_DIS
LIN {X -0.064,Y -690.864,Z 959.424,A 0.000,B 0.000,C 90.000,E1 112.333} C_DIS
LIN {X 0.055,Y -689.040,Z 959.423,A 0.000,B 0.000,C 90.000,E1 112.206} C_DIS
LIN {X -0.028,Y -683.353,Z 959.422,A 0.000,B 0.000,C 90.000,E1 111.950} C_DIS
LIN {X -0.277,Y -681.583,Z 959.422,A 0.000,B 0.000,C 90.000,E1 111.897} C_DIS
LIN {X -0.026,Y -676.295,Z 959.421,A 0.000,B 0.000,C 90.000,E1 111.716} C_DIS
LIN {X -0.272,Y -675.163,Z 959.421,A 0.000,B 0.000,C 90.000,E1 111.716} C_DIS
LIN {X -0.195,Y -667.910,Z 959.420,A 0.000,B 0.000,C 90.000,E1 111.663} C_DIS
LIN {X 0.003,Y -629.775,Z 959.420,A 0.000,B 0.000,C 90.000,E1 111.642} C_DIS
LIN {X 0.125,Y -623.607,Z 959.420,A 0.000,B 0.000,C 90.000,E1 111.535} C_DIS
LIN {X -0.281,Y -616.609,Z 959.419,A 0.000,B 0.000,C 90.000,E1 111.408} C_DIS
LIN {X -0.025,Y -609.647,Z 959.418,A 0.000,B 0.000,C 90.000,E1 111.153} C_DIS
LIN {X -0.155,Y -606.610,Z 959.417,A 0.000,B 0.000,C 90.000,E1 111.046} C_DIS
LIN {X 0.203,Y -598.679,Z 959.415,A 0.000,B 0.000,C 90.000,E1 110.610} C_DIS
LIN {X -0.303,Y -592.223,Z 959.412,A 0.000,B 0.000,C 90.000,E1 110.248} C_DIS
LIN {X 0.073,Y -576.347,Z 959.406,A 0.000,B 0.000,C 90.000,E1 109.033} C_DIS
LIN {X -0.014,Y -567.903,Z 959.403,A 0.000,B 0.000,C 90.000,E1 108.544} C_DIS
LIN {X 0.189,Y -553.253,Z 959.399,A 0.000,B 0.000,C 90.000,E1 107.819} C_DIS
LIN {X -0.076,Y -551.273,Z 959.398,A 0.000,B 0.000,C 90.000,E1 107.638} C_DIS
LIN {X -0.116,Y -551.252,Z 959.398,A 0.000,B 0.000,C 90.000,E1 107.638} C_DIS
LIN {X -0.136,Y -550.598,Z 959.397,A 0.000,B 0.000,C 90.000,E1 107.402} C_DIS
LIN {X -0.004,Y -550.617,Z 959.392,A 0.000,B 0.000,C 90.000,E1 106.551} C_DIS
LIN {X 0.077,Y -551.492,Z 959.380,A 0.000,B 0.000,C 90.000,E1 104.300} C_DIS
LIN {X -0.061,Y -552.670,Z 959.369,A 0.000,B 0.000,C 90.000,E1 102.355} C_DIS
LIN {X -0.016,Y -555.048,Z 959.353,A 0.000,B 0.000,C 90.000,E1 99.557} C_DIS
LIN {X -0.010,Y -556.338,Z 959.345,A 0.000,B 0.000,C 90.000,E1 98.163} C_DIS
LIN {X -0.060,Y -557.620,Z 959.338,A 0.000,B 0.000,C 90.000,E1 96.777} C_DIS
LIN {X -0.020,Y -558.819,Z 959.328,A 0.000,B 0.000,C 90.000,E1 95.106} C_DIS
LIN {X 0.266,Y -559.346,Z 959.324,A 0.000,B 0.000,C 90.000,E1 94.245} C_DIS
LIN {X -0.263,Y -560.306,Z 959.315,A 0.000,B 0.000,C 90.000,E1 92.636} C_DIS
LIN {X 0.220,Y -560.990,Z 959.307,A 0.000,B 0.000,C 90.000,E1 91.203} C_DIS
LIN {X 0.144,Y -561.550,Z 959.299,A 0.000,B 0.000,C 90.000,E1 89.828} C_DIS
LIN {X 0.074,Y -561.963,Z 959.292,A 0.000,B 0.000,C 90.000,E1 88.453} C_DIS
LIN {X 0.150,Y -562.358,Z 959.282,A 0.000,B 0.000,C 90.000,E1 86.788} C_DIS
LIN {X 0.106,Y -562.552,Z 959.275,A 0.000,B 0.000,C 90.000,E1 85.412} C_DIS
LIN {X 0.012,Y -562.750,Z 959.268,A 0.000,B 0.000,C 90.000,E1 84.318} C_DIS
LIN {X 0.157,Y -562.995,Z 959.259,A 0.000,B 0.000,C 90.000,E1 82.648} C_DIS
LIN {X -0.187,Y -563.345,Z 959.250,A 0.000,B 0.000,C 90.000,E1 81.027} C_DIS
LIN {X -0.104,Y -564.233,Z 959.238,A 0.000,B 0.000,C 90.000,E1 78.814} C_DIS
LIN {X -0.050,Y -565.205,Z 959.227,A 0.000,B 0.000,C 90.000,E1 76.881} C_DIS
LIN {X -0.014,Y -566.202,Z 959.218,A 0.000,B 0.000,C 90.000,E1 75.227} C_DIS
LIN {X -0.189,Y -567.546,Z 959.207,A 0.000,B 0.000,C 90.000,E1 73.323} C_DIS
LIN {X -0.126,Y -568.424,Z 959.200,A 0.000,B 0.000,C 90.000,E1 71.945} C_DIS
LIN {X -0.064,Y -569.331,Z 959.191,A 0.000,B 0.000,C 90.000,E1 70.296} C_DIS
LIN {X 0.027,Y -570.041,Z 959.181,A 0.000,B 0.000,C 90.000,E1 68.646} C_DIS
LIN {X -0.191,Y -570.310,Z 959.177,A 0.000,B 0.000,C 90.000,E1 67.847} C_DIS
LIN {X 0.118,Y -570.831,Z 959.168,A 0.000,B 0.000,C 90.000,E1 66.177} C_DIS
LIN {X -0.209,Y -571.173,Z 959.160,A 0.000,B 0.000,C 90.000,E1 64.845} C_DIS
LIN {X -0.091,Y -571.528,Z 959.150,A 0.000,B 0.000,C 90.000,E1 62.922} C_DIS
LIN {X 0.022,Y -571.643,Z 959.143,A 0.000,B 0.000,C 90.000,E1 61.820} C_DIS
LIN {X -0.034,Y -571.749,Z 959.136,A 0.000,B 0.000,C 90.000,E1 60.461} C_DIS
LIN {X 0.135,Y -571.949,Z 959.125,A 0.000,B 0.000,C 90.000,E1 58.535} C_DIS
LIN {X 0.169,Y -572.019,Z 959.118,A 0.000,B 0.000,C 90.000,E1 57.168} C_DIS
LIN {X 0.015,Y -571.683,Z 959.109,A 0.000,B 0.000,C 90.000,E1 55.548} C_DIS
LIN {X -0.109,Y -571.301,Z 959.101,A 0.000,B 0.000,C 90.000,E1 54.196} C_DIS
LIN {X 0.089,Y -570.808,Z 959.095,A 0.000,B 0.000,C 90.000,E1 53.084} C_DIS
LIN {X 0.163,Y -570.016,Z 959.089,A 0.000,B 0.000,C 90.000,E1 51.984} C_DIS
LIN {X 0.230,Y -569.061,Z 959.083,A 0.000,B 0.000,C 90.000,E1 50.884} C_DIS
LIN {X -0.154,Y -567.946,Z 959.077,A 0.000,B 0.000,C 90.000,E1 49.828} C_DIS
LIN {X -0.234,Y -566.915,Z 959.072,A 0.000,B 0.000,C 90.000,E1 49.013} C_DIS
LIN {X 0.045,Y -565.667,Z 959.068,A 0.000,B 0.000,C 90.000,E1 48.162} C_DIS
LIN {X 0.310,Y -564.225,Z 959.063,A 0.000,B 0.000,C 90.000,E1 47.310} C_DIS
LIN {X -0.237,Y -562.610,Z 959.058,A 0.000,B 0.000,C 90.000,E1 46.539} C_DIS
LIN {X -0.088,Y -561.494,Z 959.055,A 0.000,B 0.000,C 90.000,E1 45.972} C_DIS
LIN {X -0.272,Y -559.483,Z 959.051,A 0.000,B 0.000,C 90.000,E1 45.162} C_DIS
LIN {X 0.312,Y -557.220,Z 959.046,A 0.000,B 0.000,C 90.000,E1 44.271} C_DIS
LIN {X 0.079,Y -554.640,Z 959.042,A 0.000,B 0.000,C 90.000,E1 43.461} C_DIS
LIN {X -0.208,Y -552.817,Z 959.038,A 0.000,B 0.000,C 90.000,E1 42.933} C_DIS
LIN {X -0.132,Y -550.824,Z 959.035,A 0.000,B 0.000,C 90.000,E1 42.366} C_DIS
LIN {X -0.235,Y -548.068,Z 959.031,A 0.000,B 0.000,C 90.000,E1 41.676} C_DIS
LIN {X 0.029,Y -543.813,Z 959.026,A 0.000,B 0.000,C 90.000,E1 40.663} C_DIS
LIN {X 0.268,Y -540.374,Z 959.022,A 0.000,B 0.000,C 90.000,E1 39.930} C_DIS
LIN {X -0.103,Y -535.866,Z 959.017,A 0.000,B 0.000,C 90.000,E1 39.116} C_DIS
LIN {X -0.097,Y -532.733,Z 959.014,A 0.000,B 0.000,C 90.000,E1 38.543} C_DIS
LIN {X 0.027,Y -526.833,Z 959.009,A 0.000,B 0.000,C 90.000,E1 37.523} C_DIS
LIN {X -0.065,Y -521.494,Z 959.004,A 0.000,B 0.000,C 90.000,E1 36.664} C_DIS
LIN {X 0.020,Y -518.709,Z 959.001,A 0.000,B 0.000,C 90.000,E1 36.217} C_DIS
LIN {X 0.070,Y -511.942,Z 958.996,A 0.000,B 0.000,C 90.000,E1 35.185} C_DIS
LIN {X 0.010,Y -506.624,Z 958.991,A 0.000,B 0.000,C 90.000,E1 34.452} C_DIS
LIN {X 0.135,Y -503.226,Z 958.989,A 0.000,B 0.000,C 90.000,E1 33.992} C_DIS
LIN {X 0.088,Y -498.595,Z 958.986,A 0.000,B 0.000,C 90.000,E1 33.420} C_DIS
LIN {X 0.020,Y -493.483,Z 958.982,A 0.000,B 0.000,C 90.000,E1 32.832} C_DIS
LIN {X -0.222,Y -489.461,Z 958.980,A 0.000,B 0.000,C 90.000,E1 32.418} C_DIS
LIN {X -0.067,Y -484.235,Z 958.977,A 0.000,B 0.000,C 90.000,E1 31.848} C_DIS
LIN {X -0.062,Y -479.926,Z 958.975,A 0.000,B 0.000,C 90.000,E1 31.416} C_DIS
LIN {X 0.106,Y -472.844,Z 958.971,A 0.000,B 0.000,C 90.000,E1 30.718} C_DIS
LIN {X -0.009,Y -465.553,Z 958.967,A 0.000,B 0.000,C 90.000,E1 30.050} C_DIS
LIN {X 0.251,Y -455.055,Z 958.962,A 0.000,B 0.000,C 90.000,E1 29.077} C_DIS
LIN {X 0.078,Y -444.237,Z 958.957,A 0.000,B 0.000,C 90.000,E1 28.180} C_DIS
LIN {X 0.126,Y -421.377,Z 958.946,A 0.000,B 0.000,C 90.000,E1 26.181} C_DIS
LIN {X 0.186,Y -405.548,Z 958.937,A 0.000,B 0.000,C 90.000,E1 24.643} C_DIS
LIN {X 0.000,Y -398.371,Z 958.933,A 0.000,B 0.000,C 90.000,E1 23.898} C_DIS
LIN {X -0.226,Y -397.011,Z 958.932,A 0.000,B 0.000,C 90.000,E1 23.770} C_DIS
LIN {X 0.179,Y -393.887,Z 958.929,A 0.000,B 0.000,C 90.000,E1 23.259} C_DIS
LIN {X -0.017,Y -392.715,Z 958.929,A 0.000,B 0.000,C 90.000,E1 23.131} C_DIS
LIN {X 0.032,Y -391.130,Z 958.927,A 0.000,B 0.000,C 90.000,E1 22.770} C_DIS
LIN {X -0.141,Y -389.768,Z 958.923,A 0.000,B 0.000,C 90.000,E1 22.153} C_DIS
LIN {X 0.078,Y -389.474,Z 958.919,A 0.000,B 0.000,C 90.000,E1 21.408} C_DIS
LIN {X -0.037,Y -389.954,Z 958.913,A 0.000,B 0.000,C 90.000,E1 20.355} C_DIS
LIN {X -0.107,Y -392.248,Z 958.899,A 0.000,B 0.000,C 90.000,E1 17.873} C_DIS
LIN {X 0.050,Y -395.927,Z 958.882,A 0.000,B 0.000,C 90.000,E1 14.662} C_DIS
LIN {X 0.159,Y -400.292,Z 958.864,A 0.000,B 0.000,C 90.000,E1 11.478} C_DIS
LIN {X 0.114,Y -404.835,Z 958.848,A 0.000,B 0.000,C 90.000,E1 8.690} C_DIS
LIN {X 0.138,Y -409.282,Z 958.835,A 0.000,B 0.000,C 90.000,E1 6.258} C_DIS
LIN {X 0.190,Y -414.815,Z 958.820,A 0.000,B 0.000,C 90.000,E1 3.498} C_DIS
LIN {X -0.045,Y -420.939,Z 958.804,A 0.000,B 0.000,C 90.000,E1 0.802} C_DIS
LIN {X 0.000,Y -422.817,Z 958.800,A 0.000,B 0.000,C 90.000,E1 360.000} C_DIS
LIN {X -0.142,Y -424.367,Z 958.797,A 0.000,B 0.000,C 90.000,E1 359.542} C_DIS
LIN {X -0.095,Y -425.672,Z 958.796,A 0.000,B 0.000,C 90.000,E1 359.198} C_DIS
LIN {X -0.065,Y -428.298,Z 958.793,A 0.000,B 0.000,C 90.000,E1 358.682} C_DIS
LIN {X -0.034,Y -429.300,Z 958.792,A 0.000,B 0.000,C 90.000,E1 358.511} C_DIS
LIN {X -0.002,Y -430.771,Z 958.791,A 0.000,B 0.000,C 90.000,E1 358.339} C_DIS
LIN {X 0.209,Y -434.603,Z 958.789,A 0.000,B 0.000,C 90.000,E1 357.936} C_DIS
LIN {X -0.196,Y -438.946,Z 958.787,A 0.000,B 0.000,C 90.000,E1 357.707} C_DIS
LIN {X -0.095,Y -454.044,Z 958.783,A 0.000,B 0.000,C 90.000,E1 356.906} C_DIS
LIN {X 0.065,Y -470.895,Z 958.778,A 0.000,B 0.000,C 90.000,E1 355.988} C_DIS
LIN {X -0.128,Y -480.900,Z 958.775,A 0.000,B 0.000,C 90.000,E1 355.469} C_DIS
LIN {X 0.099,Y -493.912,Z 958.771,A 0.000,B 0.000,C 90.000,E1 354.723} C_DIS
LIN {X 0.229,Y -503.705,Z 958.768,A 0.000,B 0.000,C 90.000,E1 354.147} C_DIS
LIN {X 0.163,Y -513.299,Z 958.764,A 0.000,B 0.000,C 90.000,E1 353.571} C_DIS
LIN {X -0.134,Y -524.297,Z 958.760,A 0.000,B 0.000,C 90.000,E1 352.875} C_DIS
LIN {X 0.160,Y -531.791,Z 958.757,A 0.000,B 0.000,C 90.000,E1 352.299} C_DIS
LIN {X 0.087,Y -539.074,Z 958.754,A 0.000,B 0.000,C 90.000,E1 351.724} C_DIS
LIN {X -0.139,Y -545.947,Z 958.751,A 0.000,B 0.000,C 90.000,E1 351.141} C_DIS
LIN {X -0.115,Y -551.311,Z 958.748,A 0.000,B 0.000,C 90.000,E1 350.622} C_DIS
LIN {X -0.179,Y -556.470,Z 958.745,A 0.000,B 0.000,C 90.000,E1 350.095} C_DIS
LIN {X -0.109,Y -562.308,Z 958.741,A 0.000,B 0.000,C 90.000,E1 349.398} C_DIS
LIN {X 0.208,Y -566.693,Z 958.738,A 0.000,B 0.000,C 90.000,E1 348.814} C_DIS
LIN {X -0.057,Y -573.693,Z 958.733,A 0.000,B 0.000,C 90.000,E1 347.881} C_DIS
LIN {X -0.009,Y -578.990,Z 958.728,A 0.000,B 0.000,C 90.000,E1 347.061} C_DIS
LIN {X -0.006,Y -584.730,Z 958.723,A 0.000,B 0.000,C 90.000,E1 346.117} C_DIS
LIN {X 0.301,Y -589.213,Z 958.718,A 0.000,B 0.000,C 90.000,E1 345.283} C_DIS
LIN {X -0.066,Y -593.568,Z 958.714,A 0.000,B 0.000,C 90.000,E1 344.519} C_DIS
LIN {X -0.075,Y -600.112,Z 958.707,A 0.000,B 0.000,C 90.000,E1 343.196} C_DIS
LIN {X -0.124,Y -603.213,Z 958.703,A 0.000,B 0.000,C 90.000,E1 342.543} C_DIS
LIN {X -0.197,Y -606.820,Z 958.699,A 0.000,B 0.000,C 90.000,E1 341.764} C_DIS
LIN {X 0.210,Y -612.390,Z 958.691,A 0.000,B 0.000,C 90.000,E1 340.423} C_DIS
LIN {X 0.179,Y -616.560,Z 958.686,A 0.000,B 0.000,C 90.000,E1 339.390} C_DIS
LIN {X 0.196,Y -620.474,Z 958.680,A 0.000,B 0.000,C 90.000,E1 338.358} C_DIS
LIN {X -0.080,Y -623.222,Z 958.676,A 0.000,B 0.000,C 90.000,E1 337.614} C_DIS
LIN {X -0.323,Y -626.702,Z 958.670,A 0.000,B 0.000,C 90.000,E1 336.613} C_DIS
LIN {X 0.313,Y -629.940,Z 958.664,A 0.000,B 0.000,C 90.000,E1 335.537} C_DIS
LIN {X 0.160,Y -633.022,Z 958.659,A 0.000,B 0.000,C 90.000,E1 334.537} C_DIS
LIN {X 0.275,Y -635.150,Z 958.654,A 0.000,B 0.000,C 90.000,E1 333.768} C_DIS
LIN {X -0.104,Y -637.824,Z 958.649,A 0.000,B 0.000,C 90.000,E1 332.794} C_DIS
LIN {X 0.120,Y -640.283,Z 958.643,A 0.000,B 0.000,C 90.000,E1 331.769} C_DIS
LIN {X -0.131,Y -643.127,Z 958.636,A 0.000,B 0.000,C 90.000,E1 330.539} C_DIS
LIN {X -0.095,Y -645.209,Z 958.631,A 0.000,B 0.000,C 90.000,E1 329.537} C_DIS
LIN {X -0.101,Y -646.669,Z 958.627,A 0.000,B 0.000,C 90.000,E1 328.791} C_DIS
LIN {X 0.061,Y -648.751,Z 958.620,A 0.000,B 0.000,C 90.000,E1 327.533} C_DIS
LIN {X -0.023,Y -650.207,Z 958.614,A 0.000,B 0.000,C 90.000,E1 326.548} C_DIS
LIN {X 0.000,Y -651.741,Z 958.607,A 0.000,B 0.000,C 90.000,E1 325.308} C_DIS
LIN {X 0.052,Y -652.577,Z 958.603,A 0.000,B 0.000,C 90.000,E1 324.562} C_DIS
LIN {X -0.049,Y -653.768,Z 958.596,A 0.000,B 0.000,C 90.000,E1 323.336} C_DIS
LIN {X -0.124,Y -654.695,Z 958.589,A 0.000,B 0.000,C 90.000,E1 322.110} C_DIS
LIN {X 0.220,Y -655.877,Z 958.580,A 0.000,B 0.000,C 90.000,E1 320.356} C_DIS
LIN {X 0.124,Y -656.411,Z 958.574,A 0.000,B 0.000,C 90.000,E1 319.380} C_DIS
LIN {X 0.354,Y -657.716,Z 958.562,A 0.000,B 0.000,C 90.000,E1 317.148} C_DIS
LIN {X -0.239,Y -658.732,Z 958.555,A 0.000,B 0.000,C 90.000,E1 315.972} C_DIS
LIN {X -0.358,Y -659.764,Z 958.549,A 0.000,B 0.000,C 90.000,E1 314.757} C_DIS
LIN {X -0.061,Y -661.681,Z 958.536,A 0.000,B 0.000,C 90.000,E1 312.528} C_DIS
LIN {X -0.120,Y -662.984,Z 958.528,A 0.000,B 0.000,C 90.000,E1 311.067} C_DIS
LIN {X -0.145,Y -663.936,Z 958.521,A 0.000,B 0.000,C 90.000,E1 309.850} C_DIS
LIN {X -0.063,Y -664.780,Z 958.515,A 0.000,B 0.000,C 90.000,E1 308.624} C_DIS
LIN {X 0.045,Y -665.516,Z 958.508,A 0.000,B 0.000,C 90.000,E1 307.397} C_DIS
LIN {X 0.127,Y -666.076,Z 958.500,A 0.000,B 0.000,C 90.000,E1 305.931} C_DIS
LIN {X -0.106,Y -666.314,Z 958.494,A 0.000,B 0.000,C 90.000,E1 304.978} C_DIS
LIN {X -0.085,Y -667.140,Z 958.481,A 0.000,B 0.000,C 90.000,E1 302.546} C_DIS
LIN {X -0.203,Y -668.546,Z 958.467,A 0.000,B 0.000,C 90.000,E1 300.129} C_DIS
LIN {X -0.262,Y -672.693,Z 958.448,A 0.000,B 0.000,C 90.000,E1 296.744} C_DIS
LIN {X -0.166,Y -676.452,Z 958.436,A 0.000,B 0.000,C 90.000,E1 294.567} C_DIS
LIN {X 0.216,Y -678.447,Z 958.430,A 0.000,B 0.000,C 90.000,E1 293.334} C_DIS
LIN {X -0.295,Y -679.063,Z 958.427,A 0.000,B 0.000,C 90.000,E1 292.898} C_DIS
LIN {X -0.106,Y -679.259,Z 958.426,A 0.000,B 0.000,C 90.000,E1 292.642} C_DIS
LIN {X 0.016,Y -679.329,Z 958.423,A 0.000,B 0.000,C 90.000,E1 292.153} C_DIS
LIN {X 0.140,Y -678.739,Z 958.420,A 0.000,B 0.000,C 90.000,E1 291.663} C_DIS
LIN {X 0.327,Y -678.201,Z 958.419,A 0.000,B 0.000,C 90.000,E1 291.408} C_DIS
LIN {X -0.367,Y -677.066,Z 958.418,A 0.000,B 0.000,C 90.000,E1 291.227} C_DIS
LIN {X -0.255,Y -673.240,Z 958.415,A 0.000,B 0.000,C 90.000,E1 290.737} C_DIS
LIN {X -0.173,Y -672.010,Z 958.414,A 0.000,B 0.000,C 90.000,E1 290.610} C_DIS
LIN {X 0.222,Y -664.264,Z 958.412,A 0.000,B 0.000,C 90.000,E1 290.066} C_DIS
LIN {X -0.083,Y -659.796,Z 958.410,A 0.000,B 0.000,C 90.000,E1 289.812} C_DIS
LIN {X -0.017,Y -657.864,Z 958.409,A 0.000,B 0.000,C 90.000,E1 289.631} C_DIS
LIN {X -0.058,Y -657.834,Z 958.409,A 0.000,B 0.000,C 90.000,E1 289.631} C_DIS
LIN {X 0.194,Y -657.628,Z 958.409,A 0.000,B 0.000,C 90.000,E1 289.523} C_DIS
LIN {X 0.026,Y -657.765,Z 958.408,A 0.000,B 0.000,C 90.000,E1 289.396} C_DIS
LIN {X 0.125,Y -658.294,Z 958.406,A 0.000,B 0.000,C 90.000,E1 289.141} C_DIS
LIN {X -0.104,Y -660.490,Z 958.404,A 0.000,B 0.000,C 90.000,E1 288.671} C_DIS
LIN {X 0.169,Y -663.068,Z 958.401,A 0.000,B 0.000,C 90.000,E1 288.181} C_DIS
LIN {X 0.148,Y -667.923,Z 958.396,A 0.000,B 0.000,C 90.000,E1 287.330} C_DIS
LIN {X -0.071,Y -669.793,Z 958.394,A 0.000,B 0.000,C 90.000,E1 286.985} C_DIS
LIN {X -0.025,Y -672.047,Z 958.392,A 0.000,B 0.000,C 90.000,E1 286.496} C_DIS
LIN {X -0.156,Y -674.032,Z 958.389,A 0.000,B 0.000,C 90.000,E1 286.024} C_DIS
LIN {X -0.146,Y -676.346,Z 958.385,A 0.000,B 0.000,C 90.000,E1 285.300} C_DIS
LIN {X -0.297,Y -678.115,Z 958.381,A 0.000,B 0.000,C 90.000,E1 284.592} C_DIS
LIN {X 0.274,Y -679.097,Z 958.378,A 0.000,B 0.000,C 90.000,E1 284.064} C_DIS
LIN {X 0.116,Y -680.632,Z 958.373,A 0.000,B 0.000,C 90.000,E1 283.119} C_DIS
LIN {X 0.009,Y -681.471,Z 958.369,A 0.000,B 0.000,C 90.000,E1 282.411} C_DIS
LIN {X -0.203,Y -681.829,Z 958.366,A 0.000,B 0.000,C 90.000,E1 281.951} C_DIS
LIN {X -0.303,Y -681.996,Z 958.362,A 0.000,B 0.000,C 90.000,E1 281.243} C_DIS
LIN {X 0.168,Y -681.785,Z 958.360,A 0.000,B 0.000,C 90.000,E1 280.725} C_DIS
LIN {X 0.098,Y -681.360,Z 958.357,A 0.000,B 0.000,C 90.000,E1 280.254} C_DIS
LIN {X -0.097,Y -680.605,Z 958.354,A 0.000,B 0.000,C 90.000,E1 279.792} C_DIS
LIN {X -0.181,Y -679.535,Z 958.352,A 0.000,B 0.000,C 90.000,E1 279.321} C_DIS
LIN {X -0.229,Y -678.957,Z 958.350,A 0.000,B 0.000,C 90.000,E1 279.086} C_DIS
LIN {X 0.234,Y -677.413,Z 958.348,A 0.000,B 0.000,C 90.000,E1 278.568} C_DIS
LIN {X -0.043,Y -674.639,Z 958.344,A 0.000,B 0.000,C 90.000,E1 277.871} C_DIS
LIN {X -0.273,Y -672.434,Z 958.341,A 0.000,B 0.000,C 90.000,E1 277.409} C_DIS
LIN {X 0.065,Y -669.211,Z 958.338,A 0.000,B 0.000,C 90.000,E1 276.777} C_DIS
LIN {X -0.198,Y -666.393,Z 958.335,A 0.000,B 0.000,C 90.000,E1 276.315} C_DIS
LIN {X 0.179,Y -663.149,Z 958.332,A 0.000,B 0.000,C 90.000,E1 275.796} C_DIS
LIN {X -0.124,Y -659.555,Z 958.330,A 0.000,B 0.000,C 90.000,E1 275.334} C_DIS
LIN {X 0.104,Y -654.407,Z 958.326,A 0.000,B 0.000,C 90.000,E1 274.702} C_DIS
LIN {X -0.306,Y -649.960,Z 958.323,A 0.000,B 0.000,C 90.000,E1 274.245} C_DIS
LIN {X -0.123,Y -643.876,Z 958.320,A 0.000,B 0.000,C 90.000,E1 273.612} C_DIS
LIN {X 0.242,Y -638.774,Z 958.317,A 0.000,B 0.000,C 90.000,E1 273.094} C_DIS
LIN {X 0.156,Y -632.039,Z 958.314,A 0.000,B 0.000,C 90.000,E1 272.522} C_DIS
LIN {X -0.110,Y -625.074,Z 958.311,A 0.000,B 0.000,C 90.000,E1 272.007} C_DIS
LIN {X -0.121,Y -617.484,Z 958.308,A 0.000,B 0.000,C 90.000,E1 271.489} C_DIS
LIN {X -0.021,Y -611.181,Z 958.306,A 0.000,B 0.000,C 90.000,E1 271.088} C_DIS
LIN {X -0.154,Y -604.796,Z 958.304,A 0.000,B 0.000,C 90.000,E1 270.745} C_DIS
LIN {X -0.068,Y -597.940,Z 958.302,A 0.000,B 0.000,C 90.000,E1 270.401} C_DIS
LIN {X 0.283,Y -590.789,Z 958.301,A 0.000,B 0.000,C 90.000,E1 270.057} C_DIS
LIN {X -0.120,Y -583.288,Z 958.299,A 0.000,B 0.000,C 90.000,E1 269.828} C_DIS
LIN {X -0.119,Y -577.861,Z 958.298,A 0.000,B 0.000,C 90.000,E1 269.656} C_DIS
LIN {X 0.065,Y -572.112,Z 958.297,A 0.000,B 0.000,C 90.000,E1 269.484} C_DIS
LIN {X 0.219,Y -564.136,Z 958.296,A 0.000,B 0.000,C 90.000,E1 269.312} C_DIS
LIN {X -0.019,Y -557.620,Z 958.296,A 0.000,B 0.000,C 90.000,E1 269.255} C_DIS
LIN {X 0.182,Y -549.647,Z 958.296,A 0.000,B 0.000,C 90.000,E1 269.198} C_DIS
LIN {X -0.027,Y -547.142,Z 958.296,A 0.000,B 0.000,C 90.000,E1 269.198} C_DIS
LIN {X -0.068,Y -546.817,Z 958.296,A 0.000,B 0.000,C 90.000,E1 269.198} C_DIS
LIN {X -0.201,Y -543.430,Z 958.294,A 0.000,B 0.000,C 90.000,E1 268.969} C_DIS
LIN {X -0.233,Y -543.423,Z 958.294,A 0.000,B 0.000,C 90.000,E1 268.969} C_DIS
LIN {X 0.095,Y -542.692,Z 958.292,A 0.000,B 0.000,C 90.000,E1 268.453} C_DIS
LIN {X -0.245,Y -541.332,Z 958.282,A 0.000,B 0.000,C 90.000,E1 266.788} C_DIS
LIN {X -0.053,Y -539.940,Z 958.271,A 0.000,B 0.000,C 90.000,E1 264.780} C_DIS
LIN {X 0.136,Y -538.891,Z 958.263,A 0.000,B 0.000,C 90.000,E1 263.337} C_DIS
LIN {X -0.225,Y -537.813,Z 958.255,A 0.000,B 0.000,C 90.000,E1 261.951} C_DIS
LIN {X -0.119,Y -537.013,Z 958.250,A 0.000,B 0.000,C 90.000,E1 261.084} C_DIS
LIN {X 0.085,Y -535.451,Z 958.242,A 0.000,B 0.000,C 90.000,E1 259.634} C_DIS
LIN {X 0.251,Y -534.298,Z 958.238,A 0.000,B 0.000,C 90.000,E1 258.757} C_DIS
LIN {X 0.022,Y -532.253,Z 958.228,A 0.000,B 0.000,C 90.000,E1 257.061} C_DIS
LIN {X 0.060,Y -529.493,Z 958.215,A 0.000,B 0.000,C 90.000,E1 254.755} C_DIS
LIN {X -0.040,Y -527.899,Z 958.207,A 0.000,B 0.000,C 90.000,E1 253.323} C_DIS
LIN {X -0.010,Y -526.229,Z 958.199,A 0.000,B 0.000,C 90.000,E1 251.873} C_DIS
LIN {X 0.159,Y -524.035,Z 958.190,A 0.000,B 0.000,C 90.000,E1 250.115} C_DIS
LIN {X 0.137,Y -522.577,Z 958.183,A 0.000,B 0.000,C 90.000,E1 248.954} C_DIS
LIN {X -0.241,Y -520.690,Z 958.175,A 0.000,B 0.000,C 90.000,E1 247.539} C_DIS
LIN {X 0.021,Y -518.558,Z 958.167,A 0.000,B 0.000,C 90.000,E1 246.049} C_DIS
LIN {X 0.109,Y -515.857,Z 958.157,A 0.000,B 0.000,C 90.000,E1 244.280} C_DIS
LIN {X 0.014,Y -513.564,Z 958.149,A 0.000,B 0.000,C 90.000,E1 242.820} C_DIS
LIN {X 0.104,Y -511.171,Z 958.141,A 0.000,B 0.000,C 90.000,E1 241.335} C_DIS
LIN {X 0.313,Y -509.172,Z 958.134,A 0.000,B 0.000,C 90.000,E1 240.127} C_DIS
LIN {X -0.192,Y -506.929,Z 958.128,A 0.000,B 0.000,C 90.000,E1 238.997} C_DIS
LIN {X 0.076,Y -505.159,Z 958.123,A 0.000,B 0.000,C 90.000,E1 238.074} C_DIS
LIN {X 0.164,Y -503.282,Z 958.118,A 0.000,B 0.000,C 90.000,E1 237.168} C_DIS
LIN {X -0.040,Y -501.308,Z 958.113,A 0.000,B 0.000,C 90.000,E1 236.294} C_DIS
LIN {X 0.037,Y -497.159,Z 958.103,A 0.000,B 0.000,C 90.000,E1 234.482} C_DIS
LIN {X 0.056,Y -493.859,Z 958.094,A 0.000,B 0.000,C 90.000,E1 232.970} C_DIS
LIN {X 0.011,Y -489.001,Z 958.083,A 0.000,B 0.000,C 90.000,E1 230.848} C_DIS
LIN {X 0.006,Y -484.721,Z 958.072,A 0.000,B 0.000,C 90.000,E1 229.013} C_DIS
LIN {X 0.036,Y -481.260,Z 958.064,A 0.000,B 0.000,C 90.000,E1 227.472} C_DIS
LIN {X -0.117,Y -476.430,Z 958.052,A 0.000,B 0.000,C 90.000,E1 225.324} C_DIS
LIN {X -0.257,Y -472.945,Z 958.043,A 0.000,B 0.000,C 90.000,E1 223.785} C_DIS
LIN {X -0.211,Y -470.226,Z 958.036,A 0.000,B 0.000,C 90.000,E1 222.528} C_DIS
LIN {X -0.097,Y -466.855,Z 958.027,A 0.000,B 0.000,C 90.000,E1 220.943} C_DIS
LIN {X -0.045,Y -463.304,Z 958.019,A 0.000,B 0.000,C 90.000,E1 219.358} C_DIS
LIN {X 0.288,Y -459.798,Z 958.010,A 0.000,B 0.000,C 90.000,E1 217.729} C_DIS
LIN {X 0.151,Y -457.673,Z 958.005,A 0.000,B 0.000,C 90.000,E1 216.790} C_DIS
LIN {X -0.187,Y -454.131,Z 957.996,A 0.000,B 0.000,C 90.000,E1 215.231} C_DIS
LIN {X -0.138,Y -449.937,Z 957.985,A 0.000,B 0.000,C 90.000,E1 213.293} C_DIS
LIN {X -0.055,Y -445.664,Z 957.974,A 0.000,B 0.000,C 90.000,E1 211.337} C_DIS
LIN {X 0.088,Y -441.405,Z 957.963,A 0.000,B 0.000,C 90.000,E1 209.361} C_DIS
LIN {X 0.060,Y -438.559,Z 957.956,A 0.000,B 0.000,C 90.000,E1 208.052} C_DIS
LIN {X 0.000,Y -434.933,Z 957.947,A 0.000,B 0.000,C 90.000,E1 206.411} C_DIS
LIN {X 0.049,Y -432.034,Z 957.939,A 0.000,B 0.000,C 90.000,E1 205.079} C_DIS
LIN {X -0.124,Y -428.987,Z 957.932,A 0.000,B 0.000,C 90.000,E1 203.770} C_DIS
LIN {X -0.001,Y -423.659,Z 957.919,A 0.000,B 0.000,C 90.000,E1 201.408} C_DIS
LIN {X -0.107,Y -419.386,Z 957.908,A 0.000,B 0.000,C 90.000,E1 199.396} C_DIS
LIN {X 0.102,Y -414.526,Z 957.894,A 0.000,B 0.000,C 90.000,E1 196.985} C_DIS
LIN {X 0.162,Y -411.865,Z 957.887,A 0.000,B 0.000,C 90.000,E1 195.607} C_DIS
LIN {X -0.196,Y -407.743,Z 957.875,A 0.000,B 0.000,C 90.000,E1 193.592} C_DIS
LIN {X 0.044,Y -403.698,Z 957.864,A 0.000,B 0.000,C 90.000,E1 191.478} C_DIS
LIN {X 0.107,Y -400.412,Z 957.854,A 0.000,B 0.000,C 90.000,E1 189.726} C_DIS
LIN {X -0.027,Y -397.042,Z 957.844,A 0.000,B 0.000,C 90.000,E1 187.992} C_DIS
LIN {X 0.130,Y -393.085,Z 957.833,A 0.000,B 0.000,C 90.000,E1 185.853} C_DIS
LIN {X -0.054,Y -388.552,Z 957.817,A 0.000,B 0.000,C 90.000,E1 183.037} C_DIS
LIN {X 0.148,Y -387.668,Z 957.813,A 0.000,B 0.000,C 90.000,E1 182.293} C_DIS
LIN {X -0.029,Y -387.198,Z 957.809,A 0.000,B 0.000,C 90.000,E1 181.604} C_DIS
LIN {X 0.117,Y -387.142,Z 957.804,A 0.000,B 0.000,C 90.000,E1 180.688} C_DIS
LIN {X 0.068,Y -387.372,Z 957.803,A 0.000,B 0.000,C 90.000,E1 180.516} C_DIS
LIN {X -0.076,Y -387.700,Z 957.800,A 0.000,B 0.000,C 90.000,E1 180.000} C_DIS
LIN {X 0.151,Y -388.504,Z 957.798,A 0.000,B 0.000,C 90.000,E1 179.599} C_DIS
LIN {X 0.012,Y -389.379,Z 957.795,A 0.000,B 0.000,C 90.000,E1 179.083} C_DIS
LIN {X 0.013,Y -391.648,Z 957.792,A 0.000,B 0.000,C 90.000,E1 178.511} C_DIS
LIN {X -0.138,Y -393.990,Z 957.789,A 0.000,B 0.000,C 90.000,E1 178.108} C_DIS
LIN {X -0.083,Y -397.807,Z 957.787,A 0.000,B 0.000,C 90.000,E1 177.593} C_DIS
LIN {X 0.054,Y -400.639,Z 957.785,A 0.000,B 0.000,C 90.000,E1 177.249} C_DIS
LIN {X 0.162,Y -407.001,Z 957.781,A 0.000,B 0.000,C 90.000,E1 176.617} C_DIS
LIN {X 0.081,Y -424.255,Z 957.773,A 0.000,B 0.000,C 90.000,E1 175.122} C_DIS
LIN {X -0.223,Y -436.471,Z 957.767,A 0.000,B 0.000,C 90.000,E1 174.090} C_DIS
LIN {X 0.128,Y -445.359,Z 957.763,A 0.000,B 0.000,C 90.000,E1 173.223} C_DIS
LIN {X 0.047,Y -455.463,Z 957.757,A 0.000,B 0.000,C 90.000,E1 172.243} C_DIS
LIN {X 0.135,Y -461.074,Z 957.754,A 0.000,B 0.000,C 90.000,E1 171.659} C_DIS
LIN {X -0.048,Y -469.347,Z 957.749,A 0.000,B 0.000,C 90.000,E1 170.792} C_DIS
LIN {X -0.006,Y -476.005,Z 957.745,A 0.000,B 0.000,C 90.000,E1 170.038} C_DIS
LIN {X 0.259,Y -485.078,Z 957.739,A 0.000,B 0.000,C 90.000,E1 168.926} C_DIS
LIN {X 0.138,Y -491.288,Z 957.734,A 0.000,B 0.000,C 90.000,E1 168.173} C_DIS
LIN {X 0.003,Y -501.362,Z 957.727,A 0.000,B 0.000,C 90.000,E1 166.825} C_DIS
LIN {X -0.082,Y -507.701,Z 957.722,A 0.000,B 0.000,C 90.000,E1 165.936} C_DIS
LIN {X 0.107,Y -512.878,Z 957.718,A 0.000,B 0.000,C 90.000,E1 165.172} C_DIS
LIN {X -0.029,Y -519.568,Z 957.712,A 0.000,B 0.000,C 90.000,E1 164.157} C_DIS
LIN {X -0.089,Y -526.015,Z 957.706,A 0.000,B 0.000,C 90.000,E1 163.142} C_DIS
LIN {X -0.084,Y -530.447,Z 957.702,A 0.000,B 0.000,C 90.000,E1 162.417} C_DIS
LIN {X 0.209,Y -538.370,Z 957.695,A 0.000,B 0.000,C 90.000,E1 161.094} C_DIS
LIN {X 0.107,Y -546.099,Z 957.688,A 0.000,B 0.000,C 90.000,E1 159.826} C_DIS
LIN {X -0.029,Y -550.273,Z 957.684,A 0.000,B 0.000,C 90.000,E1 159.135} C_DIS
LIN {X -0.038,Y -556.006,Z 957.679,A 0.000,B 0.000,C 90.000,E1 158.156} C_DIS
LIN {X -0.087,Y -562.187,Z 957.672,A 0.000,B 0.000,C 90.000,E1 157.050} C_DIS
LIN {X -0.068,Y -565.894,Z 957.669,A 0.000,B 0.000,C 90.000,E1 156.357} C_DIS
LIN {X 0.159,Y -572.158,Z 957.662,A 0.000,B 0.000,C 90.000,E1 155.101} C_DIS
LIN {X 0.270,Y -575.474,Z 957.658,A 0.000,B 0.000,C 90.000,E1 154.409} C_DIS
LIN {X -0.095,Y -582.582,Z 957.649,A 0.000,B 0.000,C 90.000,E1 152.820} C_DIS
LIN {X -0.216,Y -585.808,Z 957.645,A 0.000,B 0.000,C 90.000,E1 152.025} C_DIS
LIN {X -0.009,Y -590.847,Z 957.637,A 0.000,B 0.000,C 90.000,E1 150.667} C_DIS
LIN {X -0.039,Y -593.613,Z 957.633,A 0.000,B 0.000,C 90.000,E1 149.871} C_DIS
LIN {X 0.081,Y -598.220,Z 957.625,A 0.000,B 0.000,C 90.000,E1 148.535} C_DIS
LIN {X 0.125,Y -600.823,Z 957.621,A 0.000,B 0.000,C 90.000,E1 147.740} C_DIS
LIN {X -0.139,Y -606.881,Z 957.611,A 0.000,B 0.000,C 90.000,E1 145.928} C_DIS
LIN {X -0.248,Y -612.962,Z 957.601,A 0.000,B 0.000,C 90.000,E1 144.116} C_DIS
LIN {X -0.025,Y -614.626,Z 957.598,A 0.000,B 0.000,C 90.000,E1 143.577} C_DIS
LIN {X 0.138,Y -618.877,Z 957.591,A 0.000,B 0.000,C 90.000,E1 142.271} C_DIS
LIN {X 0.052,Y -622.280,Z 957.585,A 0.000,B 0.000,C 90.000,E1 141.251} C_DIS
LIN {X 0.201,Y -627.211,Z 957.576,A 0.000,B 0.000,C 90.000,E1 139.703} C_DIS
LIN {X 0.029,Y -631.458,Z 957.569,A 0.000,B 0.000,C 90.000,E1 138.447} C_DIS
LIN {X -0.226,Y -637.649,Z 957.559,A 0.000,B 0.000,C 90.000,E1 136.701} C_DIS
LIN {X 0.227,Y -642.048,Z 957.552,A 0.000,B 0.000,C 90.000,E1 135.405} C_DIS
LIN {X -0.283,Y -648.267,Z 957.543,A 0.000,B 0.000,C 90.000,E1 133.704} C_DIS
LIN {X -0.044,Y -651.884,Z 957.537,A 0.000,B 0.000,C 90.000,E1 132.690} C_DIS
LIN {X 0.150,Y -659.187,Z 957.526,A 0.000,B 0.000,C 90.000,E1 130.701} C_DIS
LIN {X 0.077,Y -663.856,Z 957.519,A 0.000,B 0.000,C 90.000,E1 129.483} C_DIS
LIN {X 0.158,Y -669.309,Z 957.511,A 0.000,B 0.000,C 90.000,E1 128.016} C_DIS
LIN {X 0.345,Y -673.613,Z 957.505,A 0.000,B 0.000,C 90.000,E1 126.790} C_DIS
LIN {X -0.341,Y -676.951,Z 957.499,A 0.000,B 0.000,C 90.000,E1 125.884} C_DIS
LIN {X -0.041,Y -680.768,Z 957.493,A 0.000,B 0.000,C 90.000,E1 124.659} C_DIS
LIN {X -0.078,Y -683.685,Z 957.487,A 0.000,B 0.000,C 90.000,E1 123.706} C_DIS
LIN {X 0.133,Y -686.892,Z 957.481,A 0.000,B 0.000,C 90.000,E1 122.498} C_DIS
LIN {X -0.182,Y -689.920,Z 957.474,A 0.000,B 0.000,C 90.000,E1 121.337} C_DIS
LIN {X 0.261,Y -691.562,Z 957.470,A 0.000,B 0.000,C 90.000,E1 120.590} C_DIS
LIN {X 0.008,Y -693.444,Z 957.465,A 0.000,B 0.000,C 90.000,E1 119.667} C_DIS
LIN {X -0.110,Y -694.307,Z 957.462,A 0.000,B 0.000,C 90.000,E1 119.205} C_DIS
LIN {X 0.279,Y -695.630,Z 957.457,A 0.000,B 0.000,C 90.000,E1 118.231} C_DIS
LIN {X 0.067,Y -696.687,Z 957.452,A 0.000,B 0.000,C 90.000,E1 117.308} C_DIS
LIN {X -0.197,Y -697.500,Z 957.445,A 0.000,B 0.000,C 90.000,E1 116.155} C_DIS
LIN {X 0.178,Y -697.936,Z 957.439,A 0.000,B 0.000,C 90.000,E1 114.951} C_DIS
LIN {X 0.037,Y -698.056,Z 957.435,A 0.000,B 0.000,C 90.000,E1 114.259} C_DIS
LIN {X 0.275,Y -697.792,Z 957.432,A 0.000,B 0.000,C 90.000,E1 113.770} C_DIS
LIN {X -0.105,Y -697.289,Z 957.431,A 0.000,B 0.000,C 90.000,E1 113.567} C_DIS
LIN {X 0.133,Y -695.950,Z 957.428,A 0.000,B 0.000,C 90.000,E1 113.078} C_DIS
LIN {X 0.259,Y -695.345,Z 957.428,A 0.000,B 0.000,C 90.000,E1 112.950} C_DIS
LIN {X -0.156,Y -692.241,Z 957.425,A 0.000,B 0.000,C 90.000,E1 112.514} C_DIS
LIN {X -0.036,Y -691.241,Z 957.424,A 0.000,B 0.000,C 90.000,E1 112.386} C_DIS
LIN {X -0.181,Y -689.740,Z 957.424,A 0.000,B 0.000,C 90.000,E1 112.280} C_DIS
LIN {X -0.152,Y -685.875,Z 957.423,A 0.000,B 0.000,C 90.000,E1 112.078} C_DIS
LIN {X -0.056,Y -680.647,Z 957.421,A 0.000,B 0.000,C 90.000,E1 111.844} C_DIS
LIN {X -0.170,Y -675.878,Z 957.421,A 0.000,B 0.000,C 90.000,E1 111.716} C_DIS
LIN {X 0.202,Y -674.150,Z 957.420,A 0.000,B 0.000,C 90.000,E1 111.663} C_DIS
LIN {X -0.060,Y -667.477,Z 957.420,A 0.000,B 0.000,C 90.000,E1 111.642} C_DIS
LIN {X -0.093,Y -630.482,Z 957.420,A 0.000,B 0.000,C 90.000,E1 111.642} C_DIS
LIN {X -0.241,Y -625.819,Z 957.420,A 0.000,B 0.000,C 90.000,E1 111.589} C_DIS
LIN {X -0.316,Y -622.326,Z 957.420,A 0.000,B 0.000,C 90.000,E1 111.535} C_DIS
LIN {X 0.231,Y -617.155,Z 957.419,A 0.000,B 0.000,C 90.000,E1 111.354} C_DIS
LIN {X -0.106,Y -610.050,Z 957.417,A 0.000,B 0.000,C 90.000,E1 111.153} C_DIS
LIN {X 0.136,Y -606.039,Z 957.417,A 0.000,B 0.000,C 90.000,E1 110.972} C_DIS
LIN {X -0.270,Y -600.599,Z 957.415,A 0.000,B 0.000,C 90.000,E1 110.737} C_DIS
LIN {X 0.120,Y -593.944,Z 957.413,A 0.000,B 0.000,C 90.000,E1 110.301} C_DIS
LIN {X -0.134,Y -576.095,Z 957.406,A 0.000,B 0.000,C 90.000,E1 109.014} C_DIS
LIN {X -0.235,Y -567.715,Z 957.403,A 0.000,B 0.000,C 90.000,E1 108.544} C_DIS
LIN {X 0.050,Y -554.237,Z 957.399,A 0.000,B 0.000,C 90.000,E1 107.873} C_DIS
LIN {X -0.166,Y -552.931,Z 957.399,A 0.000,B 0.000,C 90.000,E1 107.819} C_DIS
LIN {X 0.102,Y -551.481,Z 957.398,A 0.000,B 0.000,C 90.000,E1 107.638} C_DIS
LIN {X 0.058,Y -551.440,Z 957.398,A 0.000,B 0.000,C 90.000,E1 107.638} C_DIS
LIN {X 0.061,Y -550.703,Z 957.396,A 0.000,B 0.000,C 90.000,E1 107.330} C_DIS
LIN {X -0.092,Y -550.798,Z 957.391,A 0.000,B 0.000,C 90.000,E1 106.370} C_DIS
LIN {X 0.165,Y -551.455,Z 957.382,A 0.000,B 0.000,C 90.000,E1 104.662} C_DIS
LIN {X -0.145,Y -552.929,Z 957.368,A 0.000,B 0.000,C 90.000,E1 102.175} C_DIS
LIN {X -0.101,Y -555.315,Z 957.352,A 0.000,B 0.000,C 90.000,E1 99.378} C_DIS
LIN {X -0.175,Y -556.595,Z 957.344,A 0.000,B 0.000,C 90.000,E1 97.992} C_DIS
LIN {X 0.273,Y -557.616,Z 957.338,A 0.000,B 0.000,C 90.000,E1 96.834} C_DIS
LIN {X -0.017,Y -558.242,Z 957.334,A 0.000,B 0.000,C 90.000,E1 96.030} C_DIS
LIN {X -0.041,Y -559.203,Z 957.326,A 0.000,B 0.000,C 90.000,E1 94.645} C_DIS
LIN {X 0.069,Y -560.315,Z 957.315,A 0.000,B 0.000,C 90.000,E1 92.694} C_DIS
LIN {X -0.009,Y -561.016,Z 957.307,A 0.000,B 0.000,C 90.000,E1 91.318} C_DIS
LIN {X -0.085,Y -561.572,Z 957.300,A 0.000,B 0.000,C 90.000,E1 89.943} C_DIS
LIN {X -0.154,Y -561.970,Z 957.292,A 0.000,B 0.000,C 90.000,E1 88.568} C_DIS
LIN {X -0.108,Y -562.392,Z 957.283,A 0.000,B 0.000,C 90.000,E1 86.906} C_DIS
LIN {X -0.119,Y -562.613,Z 957.275,A 0.000,B 0.000,C 90.000,E1 85.527} C_DIS
LIN {X -0.122,Y -562.805,Z 957.267,A 0.000,B 0.000,C 90.000,E1 84.147} C_DIS
LIN {X 0.091,Y -563.054,Z 957.258,A 0.000,B 0.000,C 90.000,E1 82.470} C_DIS
LIN {X 0.156,Y -563.392,Z 957.251,A 0.000,B 0.000,C 90.000,E1 81.084} C_DIS
LIN {X -0.145,Y -564.351,Z 957.237,A 0.000,B 0.000,C 90.000,E1 78.634} C_DIS
LIN {X -0.083,Y -565.350,Z 957.226,A 0.000,B 0.000,C 90.000,E1 76.700} C_DIS
LIN {X -0.039,Y -566.372,Z 957.217,A 0.000,B 0.000,C 90.000,E1 75.046} C_DIS
LIN {X 0.174,Y -567.509,Z 957.208,A 0.000,B 0.000,C 90.000,E1 73.378} C_DIS
LIN {X 0.240,Y -568.403,Z 957.200,A 0.000,B 0.000,C 90.000,E1 72.000} C_DIS
LIN {X -0.227,Y -569.174,Z 957.193,A 0.000,B 0.000,C 90.000,E1 70.678} C_DIS
LIN {X -0.112,Y -569.640,Z 957.187,A 0.000,B 0.000,C 90.000,E1 69.571} C_DIS
LIN {X -0.164,Y -570.214,Z 957.179,A 0.000,B 0.000,C 90.000,E1 68.209} C_DIS
LIN {X 0.152,Y -570.694,Z 957.170,A 0.000,B 0.000,C 90.000,E1 66.538} C_DIS
LIN {X -0.061,Y -571.114,Z 957.161,A 0.000,B 0.000,C 90.000,E1 64.921} C_DIS
LIN {X 0.046,Y -571.467,Z 957.150,A 0.000,B 0.000,C 90.000,E1 62.999} C_DIS
LIN {X 0.154,Y -571.589,Z 957.144,A 0.000,B 0.000,C 90.000,E1 61.897} C_DIS
LIN {X 0.206,Y -571.672,Z 957.135,A 0.000,B 0.000,C 90.000,E1 60.255} C_DIS
LIN {X -0.110,Y -571.886,Z 957.124,A 0.000,B 0.000,C 90.000,E1 58.377} C_DIS
LIN {X 0.099,Y -571.915,Z 957.117,A 0.000,B 0.000,C 90.000,E1 56.993} C_DIS
LIN {X -0.217,Y -571.501,Z 957.108,A 0.000,B 0.000,C 90.000,E1 55.388} C_DIS
LIN {X 0.125,Y -571.113,Z 957.100,A 0.000,B 0.000,C 90.000,E1 53.989} C_DIS
LIN {X -0.271,Y -570.712,Z 957.096,A 0.000,B 0.000,C 90.000,E1 53.210} C_DIS
LIN {X -0.194,Y -569.890,Z 957.089,A 0.000,B 0.000,C 90.000,E1 52.110} C_DIS
LIN {X -0.123,Y -568.938,Z 957.083,A 0.000,B 0.000,C 90.000,E1 51.009} C_DIS
LIN {X -0.068,Y -567.826,Z 957.077,A 0.000,B 0.000,C 90.000,E1 49.908} C_DIS
LIN {X -0.152,Y -566.811,Z 957.073,A 0.000,B 0.000,C 90.000,E1 49.094} C_DIS
LIN {X 0.125,Y -565.552,Z 957.068,A 0.000,B 0.000,C 90.000,E1 48.243} C_DIS
LIN {X 0.070,Y -563.557,Z 957.062,A 0.000,B 0.000,C 90.000,E1 47.148} C_DIS
LIN {X -0.012,Y -561.330,Z 957.056,A 0.000,B 0.000,C 90.000,E1 46.053} C_DIS
LIN {X -0.199,Y -559.363,Z 957.051,A 0.000,B 0.000,C 90.000,E1 45.243} C_DIS
LIN {X -0.015,Y -557.053,Z 957.047,A 0.000,B 0.000,C 90.000,E1 44.393} C_DIS
LIN {X 0.149,Y -554.482,Z 957.042,A 0.000,B 0.000,C 90.000,E1 43.542} C_DIS
LIN {X 0.290,Y -551.647,Z 957.037,A 0.000,B 0.000,C 90.000,E1 42.690} C_DIS
LIN {X -0.014,Y -549.573,Z 957.034,A 0.000,B 0.000,C 90.000,E1 42.162} C_DIS
LIN {X 0.036,Y -547.299,Z 957.031,A 0.000,B 0.000,C 90.000,E1 41.595} C_DIS
LIN {X 0.124,Y -542.322,Z 957.025,A 0.000,B 0.000,C 90.000,E1 40.458} C_DIS
LIN {X -0.227,Y -537.952,Z 957.020,A 0.000,B 0.000,C 90.000,E1 39.644} C_DIS
LIN {X 0.134,Y -533.327,Z 957.015,A 0.000,B 0.000,C 90.000,E1 38.749} C_DIS
LIN {X 0.087,Y -526.561,Z 957.009,A 0.000,B 0.000,C 90.000,E1 37.604} C_DIS
LIN {X 0.126,Y -520.287,Z 957.003,A 0.000,B 0.000,C 90.000,E1 36.583} C_DIS
LIN {X -0.041,Y -514.533,Z 956.998,A 0.000,B 0.000,C 90.000,E1 35.724} C_DIS
LIN {X -0.294,Y -511.597,Z 956.996,A 0.000,B 0.000,C 90.000,E1 35.311} C_DIS
LIN {X 0.054,Y -506.233,Z 956.992,A 0.000,B 0.000,C 90.000,E1 34.532} C_DIS
LIN {X -0.239,Y -502.836,Z 956.989,A 0.000,B 0.000,C 90.000,E1 34.119} C_DIS
LIN {X -0.257,Y -496.676,Z 956.985,A 0.000,B 0.000,C 90.000,E1 33.372} C_DIS
LIN {X 0.089,Y -492.768,Z 956.983,A 0.000,B 0.000,C 90.000,E1 32.880} C_DIS
LIN {X -0.175,Y -488.735,Z 956.980,A 0.000,B 0.000,C 90.000,E1 32.467} C_DIS
LIN {X -0.075,Y -483.198,Z 956.977,A 0.000,B 0.000,C 90.000,E1 31.878} C_DIS
LIN {X 0.186,Y -474.571,Z 956.972,A 0.000,B 0.000,C 90.000,E1 31.003} C_DIS
LIN {X 0.131,Y -465.902,Z 956.968,A 0.000,B 0.000,C 90.000,E1 30.207} C_DIS
LIN {X 0.181,Y -455.715,Z 956.963,A 0.000,B 0.000,C 90.000,E1 29.283} C_DIS
LIN {X -0.058,Y -443.588,Z 956.957,A 0.000,B 0.000,C 90.000,E1 28.281} C_DIS
LIN {X -0.082,Y -417.893,Z 956.945,A 0.000,B 0.000,C 90.000,E1 26.027} C_DIS
LIN {X -0.086,Y -403.064,Z 956.936,A 0.000,B 0.000,C 90.000,E1 24.567} C_DIS
LIN {X 0.117,Y -398.801,Z 956.934,A 0.000,B 0.000,C 90.000,E1 24.079} C_DIS
LIN {X -0.098,Y -396.387,Z 956.932,A 0.000,B 0.000,C 90.000,E1 23.823} C_DIS
LIN {X -0.071,Y -391.950,Z 956.928,A 0.000,B 0.000,C 90.000,E1 23.131} C_DIS
LIN {X 0.190,Y -390.893,Z 956.927,A 0.000,B 0.000,C 90.000,E1 22.823} C_DIS
LIN {X 0.211,Y -390.381,Z 956.926,A 0.000,B 0.000,C 90.000,E1 22.642} C_DIS
LIN {X -0.113,Y -389.739,Z 956.924,A 0.000,B 0.000,C 90.000,E1 22.333} C_DIS
LIN {X -0.039,Y -389.458,Z 956.920,A 0.000,B 0.000,C 90.000,E1 21.589} C_DIS
LIN {X -0.119,Y -390.184,Z 956.912,A 0.000,B 0.000,C 90.000,E1 20.174} C_DIS
LIN {X -0.083,Y -393.302,Z 956.894,A 0.000,B 0.000,C 90.000,E1 16.968} C_DIS
LIN {X -0.015,Y -396.276,Z 956.880,A 0.000,B 0.000,C 90.000,E1 14.481} C_DIS
LIN {X 0.100,Y -400.701,Z 956.863,A 0.000,B 0.000,C 90.000,E1 11.299} C_DIS
LIN {X 0.059,Y -405.278,Z 956.847,A 0.000,B 0.000,C 90.000,E1 8.511} C_DIS
LIN {X 0.040,Y -409.718,Z 956.834,A 0.000,B 0.000,C 90.000,E1 6.087} C_DIS
LIN {X 0.111,Y -415.309,Z 956.819,A 0.000,B 0.000,C 90.000,E1 3.326} C_DIS
LIN {X -0.071,Y -422.287,Z 956.802,A 0.000,B 0.000,C 90.000,E1 0.286} C_DIS
LIN {X 0.160,Y -423.460,Z 956.799,A 0.000,B 0.000,C 90.000,E1 359.771} C_DIS
LIN {X -0.194,Y -425.165,Z 956.796,A 0.000,B 0.000,C 90.000,E1 359.312} C_DIS
LIN {X -0.196,Y -427.843,Z 956.793,A 0.000,B 0.000,C 90.000,E1 358.740} C_DIS
LIN {X -0.168,Y -428.665,Z 956.792,A 0.000,B 0.000,C 90.000,E1 358.568} C_DIS
LIN {X -0.136,Y -429.872,Z 956.791,A 0.000,B 0.000,C 90.000,E1 358.396} C_DIS
LIN {X 0.180,Y -433.214,Z 956.789,A 0.000,B 0.000,C 90.000,E1 357.993} C_DIS
LIN {X -0.081,Y -434.848,Z 956.788,A 0.000,B 0.000,C 90.000,E1 357.879} C_DIS
LIN {X -0.193,Y -440.521,Z 956.786,A 0.000,B 0.000,C 90.000,E1 357.535} C_DIS
LIN {X -0.040,Y -453.663,Z 956.782,A 0.000,B 0.000,C 90.000,E1 356.846} C_DIS
LIN {X 0.219,Y -467.091,Z 956.779,A 0.000,B 0.000,C 90.000,E1 356.102} C_DIS
LIN {X 0.140,Y -480.151,Z 956.775,A 0.000,B 0.000,C 90.000,E1 355.412} C_DIS
LIN {X 0.135,Y -494.641,Z 956.770,A 0.000,B 0.000,C 90.000,E1 354.609} C_DIS
LIN {X -0.261,Y -504.451,Z 956.767,A 0.000,B 0.000,C 90.000,E1 354.090} C_DIS
LIN {X 0.042,Y -512.576,Z 956.764,A 0.000,B 0.000,C 90.000,E1 353.571} C_DIS
LIN {X -0.205,Y -523.452,Z 956.760,A 0.000,B 0.000,C 90.000,E1 352.875} C_DIS
LIN {X 0.109,Y -529.501,Z 956.758,A 0.000,B 0.000,C 90.000,E1 352.413} C_DIS
LIN {X 0.153,Y -536.944,Z 956.755,A 0.000,B 0.000,C 90.000,E1 351.837} C_DIS
LIN {X 0.045,Y -543.888,Z 956.751,A 0.000,B 0.000,C 90.000,E1 351.254} C_DIS
LIN {X 0.030,Y -550.627,Z 956.748,A 0.000,B 0.000,C 90.000,E1 350.622} C_DIS
LIN {X -0.015,Y -555.795,Z 956.745,A 0.000,B 0.000,C 90.000,E1 350.095} C_DIS
LIN {X 0.086,Y -561.677,Z 956.741,A 0.000,B 0.000,C 90.000,E1 349.398} C_DIS
LIN {X -0.157,Y -566.119,Z 956.738,A 0.000,B 0.000,C 90.000,E1 348.870} C_DIS
LIN {X 0.130,Y -573.215,Z 956.733,A 0.000,B 0.000,C 90.000,E1 347.881} C_DIS
LIN {X 0.175,Y -578.589,Z 956.728,A 0.000,B 0.000,C 90.000,E1 347.061} C_DIS
LIN {X -0.156,Y -583.571,Z 956.724,A 0.000,B 0.000,C 90.000,E1 346.284} C_DIS
LIN {X -0.004,Y -588.225,Z 956.719,A 0.000,B 0.000,C 90.000,E1 345.463} C_DIS
LIN {X 0.037,Y -594.004,Z 956.713,A 0.000,B 0.000,C 90.000,E1 344.393} C_DIS
LIN {X -0.132,Y -600.547,Z 956.706,A 0.000,B 0.000,C 90.000,E1 343.087} C_DIS
LIN {X 0.002,Y -603.632,Z 956.702,A 0.000,B 0.000,C 90.000,E1 342.417} C_DIS
LIN {X -0.101,Y -607.798,Z 956.697,A 0.000,B 0.000,C 90.000,E1 341.511} C_DIS
LIN {X -0.192,Y -612.277,Z 956.691,A 0.000,B 0.000,C 90.000,E1 340.477} C_DIS
LIN {X -0.224,Y -616.496,Z 956.686,A 0.000,B 0.000,C 90.000,E1 339.444} C_DIS
LIN {X -0.206,Y -620.417,Z 956.680,A 0.000,B 0.000,C 90.000,E1 338.411} C_DIS
LIN {X 0.095,Y -623.205,Z 956.676,A 0.000,B 0.000,C 90.000,E1 337.614} C_DIS
LIN {X -0.148,Y -626.700,Z 956.670,A 0.000,B 0.000,C 90.000,E1 336.613} C_DIS
LIN {X -0.345,Y -629.987,Z 956.664,A 0.000,B 0.000,C 90.000,E1 335.613} C_DIS
LIN {X -0.234,Y -633.096,Z 956.659,A 0.000,B 0.000,C 90.000,E1 334.588} C_DIS
LIN {X -0.116,Y -635.250,Z 956.655,A 0.000,B 0.000,C 90.000,E1 333.819} C_DIS
LIN {X 0.131,Y -638.597,Z 956.648,A 0.000,B 0.000,C 90.000,E1 332.538} C_DIS
LIN {X -0.200,Y -641.006,Z 956.642,A 0.000,B 0.000,C 90.000,E1 331.563} C_DIS
LIN {X 0.123,Y -643.866,Z 956.635,A 0.000,B 0.000,C 90.000,E1 330.284} C_DIS
LIN {X -0.316,Y -646.416,Z 956.628,A 0.000,B 0.000,C 90.000,E1 329.076} C_DIS
LIN {X 0.183,Y -648.572,Z 956.621,A 0.000,B 0.000,C 90.000,E1 327.788} C_DIS
LIN {X -0.256,Y -650.117,Z 956.616,A 0.000,B 0.000,C 90.000,E1 326.834} C_DIS
LIN {X 0.225,Y -651.402,Z 956.610,A 0.000,B 0.000,C 90.000,E1 325.801} C_DIS
LIN {X -0.273,Y -652.886,Z 956.603,A 0.000,B 0.000,C 90.000,E1 324.609} C_DIS
LIN {X 0.164,Y -654.053,Z 956.596,A 0.000,B 0.000,C 90.000,E1 323.336} C_DIS
LIN {X 0.094,Y -655.017,Z 956.590,A 0.000,B 0.000,C 90.000,E1 322.110} C_DIS
LIN {X -0.059,Y -656.223,Z 956.580,A 0.000,B 0.000,C 90.000,E1 320.400} C_DIS
LIN {X -0.151,Y -657.105,Z 956.572,A 0.000,B 0.000,C 90.000,E1 318.933} C_DIS
LIN {X 0.011,Y -659.128,Z 956.555,A 0.000,B 0.000,C 90.000,E1 315.972} C_DIS
LIN {X -0.101,Y -660.163,Z 956.549,A 0.000,B 0.000,C 90.000,E1 314.757} C_DIS
LIN {X 0.227,Y -661.858,Z 956.538,A 0.000,B 0.000,C 90.000,E1 312.771} C_DIS
LIN {X 0.175,Y -663.179,Z 956.530,A 0.000,B 0.000,C 90.000,E1 311.310} C_DIS
LIN {X 0.141,Y -664.377,Z 956.521,A 0.000,B 0.000,C 90.000,E1 309.850} C_DIS
LIN {X 0.230,Y -665.242,Z 956.515,A 0.000,B 0.000,C 90.000,E1 308.624} C_DIS
LIN {X 0.249,Y -665.863,Z 956.509,A 0.000,B 0.000,C 90.000,E1 307.649} C_DIS
LIN {X -0.033,Y -666.378,Z 956.503,A 0.000,B 0.000,C 90.000,E1 306.457} C_DIS
LIN {X 0.090,Y -666.776,Z 956.496,A 0.000,B 0.000,C 90.000,E1 305.231} C_DIS
LIN {X 0.250,Y -667.670,Z 956.481,A 0.000,B 0.000,C 90.000,E1 302.546} C_DIS
LIN {X -0.005,Y -668.895,Z 956.469,A 0.000,B 0.000,C 90.000,E1 300.384} C_DIS
LIN {X 0.022,Y -671.692,Z 956.454,A 0.000,B 0.000,C 90.000,E1 297.719} C_DIS
LIN {X 0.288,Y -675.592,Z 956.441,A 0.000,B 0.000,C 90.000,E1 295.283} C_DIS
LIN {X 0.132,Y -677.311,Z 956.435,A 0.000,B 0.000,C 90.000,E1 294.335} C_DIS
LIN {X -0.007,Y -678.881,Z 956.430,A 0.000,B 0.000,C 90.000,E1 293.387} C_DIS
LIN {X 0.300,Y -679.739,Z 956.426,A 0.000,B 0.000,C 90.000,E1 292.642} C_DIS
LIN {X -0.206,Y -679.764,Z 956.423,A 0.000,B 0.000,C 90.000,E1 292.206} C_DIS
LIN {X -0.016,Y -679.596,Z 956.422,A 0.000,B 0.000,C 90.000,E1 291.950} C_DIS
LIN {X -0.080,Y -679.173,Z 956.421,A 0.000,B 0.000,C 90.000,E1 291.716} C_DIS
LIN {X 0.107,Y -678.570,Z 956.419,A 0.000,B 0.000,C 90.000,E1 291.461} C_DIS
LIN {X 0.045,Y -677.617,Z 956.418,A 0.000,B 0.000,C 90.000,E1 291.227} C_DIS
LIN {X 0.071,Y -674.801,Z 956.416,A 0.000,B 0.000,C 90.000,E1 290.865} C_DIS
LIN {X 0.241,Y -672.335,Z 956.415,A 0.000,B 0.000,C 90.000,E1 290.610} C_DIS
LIN {X 0.323,Y -670.736,Z 956.414,A 0.000,B 0.000,C 90.000,E1 290.482} C_DIS
LIN {X -0.196,Y -660.412,Z 956.410,A 0.000,B 0.000,C 90.000,E1 289.866} C_DIS
LIN {X -0.170,Y -658.363,Z 956.409,A 0.000,B 0.000,C 90.000,E1 289.685} C_DIS
LIN {X -0.215,Y -658.331,Z 956.409,A 0.000,B 0.000,C 90.000,E1 289.685} C_DIS
LIN {X 0.051,Y -658.207,Z 956.408,A 0.000,B 0.000,C 90.000,E1 289.504} C_DIS
LIN {X -0.116,Y -658.412,Z 956.408,A 0.000,B 0.000,C 90.000,E1 289.396} C_DIS
LIN {X 0.278,Y -659.136,Z 956.406,A 0.000,B 0.000,C 90.000,E1 289.087} C_DIS
LIN {X -0.239,Y -662.175,Z 956.403,A 0.000,B 0.000,C 90.000,E1 288.489} C_DIS
LIN {X -0.269,Y -667.045,Z 956.398,A 0.000,B 0.000,C 90.000,E1 287.638} C_DIS
LIN {X -0.235,Y -669.704,Z 956.395,A 0.000,B 0.000,C 90.000,E1 287.149} C_DIS
LIN {X 0.192,Y -673.019,Z 956.391,A 0.000,B 0.000,C 90.000,E1 286.386} C_DIS
LIN {X 0.255,Y -674.939,Z 956.388,A 0.000,B 0.000,C 90.000,E1 285.898} C_DIS
LIN {X 0.093,Y -677.146,Z 956.384,A 0.000,B 0.000,C 90.000,E1 285.190} C_DIS
LIN {X 0.000,Y -678.344,Z 956.382,A 0.000,B 0.000,C 90.000,E1 284.717} C_DIS
LIN {X -0.125,Y -679.763,Z 956.378,A 0.000,B 0.000,C 90.000,E1 284.008} C_DIS
LIN {X -0.236,Y -680.958,Z 956.374,A 0.000,B 0.000,C 90.000,E1 283.300} C_DIS
LIN {X -0.304,Y -681.612,Z 956.371,A 0.000,B 0.000,C 90.000,E1 282.827} C_DIS
LIN {X 0.263,Y -682.314,Z 956.367,A 0.000,B 0.000,C 90.000,E1 282.063} C_DIS
LIN {X 0.231,Y -682.499,Z 956.366,A 0.000,B 0.000,C 90.000,E1 281.827} C_DIS
LIN {X 0.031,Y -682.643,Z 956.363,A 0.000,B 0.000,C 90.000,E1 281.366} C_DIS
LIN {X -0.066,Y -682.361,Z 956.359,A 0.000,B 0.000,C 90.000,E1 280.658} C_DIS
LIN {X -0.258,Y -681.937,Z 956.357,A 0.000,B 0.000,C 90.000,E1 280.197} C_DIS
LIN {X 0.338,Y -681.123,Z 956.354,A 0.000,B 0.000,C 90.000,E1 279.670} C_DIS
LIN {X 0.098,Y -679.323,Z 956.350,A 0.000,B 0.000,C 90.000,E1 278.973} C_DIS
LIN {X -0.105,Y -677.769,Z 956.347,A 0.000,B 0.000,C 90.000,E1 278.511} C_DIS
LIN {X -0.314,Y -675.921,Z 956.345,A 0.000,B 0.000,C 90.000,E1 278.049} C_DIS
LIN {X 0.135,Y -673.776,Z 956.342,A 0.000,B 0.000,C 90.000,E1 277.530} C_DIS
LIN {X -0.178,Y -670.009,Z 956.338,A 0.000,B 0.000,C 90.000,E1 276.834} C_DIS
LIN {X 0.227,Y -667.219,Z 956.335,A 0.000,B 0.000,C 90.000,E1 276.315} C_DIS
LIN {X -0.051,Y -664.085,Z 956.333,A 0.000,B 0.000,C 90.000,E1 275.853} C_DIS
LIN {X 0.214,Y -659.522,Z 956.329,A 0.000,B 0.000,C 90.000,E1 275.220} C_DIS
LIN {X -0.114,Y -655.457,Z 956.326,A 0.000,B 0.000,C 90.000,E1 274.759} C_DIS
LIN {X -0.296,Y -651.276,Z 956.324,A 0.000,B 0.000,C 90.000,E1 274.302} C_DIS
LIN {X -0.102,Y -645.259,Z 956.320,A 0.000,B 0.000,C 90.000,E1 273.669} C_DIS
LIN {X 0.235,Y -638.896,Z 956.317,A 0.000,B 0.000,C 90.000,E1 273.037} C_DIS
LIN {X 0.099,Y -632.115,Z 956.314,A 0.000,B 0.000,C 90.000,E1 272.465} C_DIS
LIN {X -0.240,Y -625.035,Z 956.311,A 0.000,B 0.000,C 90.000,E1 271.949} C_DIS
LIN {X -0.218,Y -617.461,Z 956.308,A 0.000,B 0.000,C 90.000,E1 271.432} C_DIS
LIN {X -0.052,Y -611.153,Z 956.306,A 0.000,B 0.000,C 90.000,E1 271.031} C_DIS
LIN {X -0.175,Y -604.847,Z 956.304,A 0.000,B 0.000,C 90.000,E1 270.688} C_DIS
LIN {X -0.101,Y -598.008,Z 956.302,A 0.000,B 0.000,C 90.000,E1 270.344} C_DIS
LIN {X 0.285,Y -590.939,Z 956.300,A 0.000,B 0.000,C 90.000,E1 270.000} C_DIS
LIN {X -0.128,Y -583.425,Z 956.299,A 0.000,B 0.000,C 90.000,E1 269.771} C_DIS
LIN {X -0.142,Y -577.984,Z 956.298,A 0.000,B 0.000,C 90.000,E1 269.599} C_DIS
LIN {X 0.058,Y -572.154,Z 956.297,A 0.000,B 0.000,C 90.000,E1 269.427} C_DIS
LIN {X 0.174,Y -564.178,Z 956.296,A 0.000,B 0.000,C 90.000,E1 269.255} C_DIS
LIN {X -0.069,Y -557.059,Z 956.296,A 0.000,B 0.000,C 90.000,E1 269.198} C_DIS
LIN {X 0.137,Y -550.141,Z 956.295,A 0.000,B 0.000,C 90.000,E1 269.141} C_DIS
LIN {X -0.040,Y -548.255,Z 956.295,A 0.000,B 0.000,C 90.000,E1 269.141} C_DIS
LIN {X -0.070,Y -548.073,Z 956.295,A 0.000,B 0.000,C 90.000,E1 269.141} C_DIS
LIN {X 0.101,Y -543.559,Z 956.293,A 0.000,B 0.000,C 90.000,E1 268.797} C_DIS
LIN {X 0.068,Y -543.514,Z 956.293,A 0.000,B 0.000,C 90.000,E1 268.797} C_DIS
LIN {X 0.152,Y -542.752,Z 956.291,A 0.000,B 0.000,C 90.000,E1 268.396} C_DIS
LIN {X 0.114,Y -541.453,Z 956.282,A 0.000,B 0.000,C 90.000,E1 266.788} C_DIS
LIN {X -0.231,Y -540.023,Z 956.271,A 0.000,B 0.000,C 90.000,E1 264.837} C_DIS
LIN {X -0.038,Y -538.985,Z 956.263,A 0.000,B 0.000,C 90.000,E1 263.394} C_DIS
LIN {X 0.136,Y -537.963,Z 956.255,A 0.000,B 0.000,C 90.000,E1 261.951} C_DIS
LIN {X -0.226,Y -536.886,Z 956.249,A 0.000,B 0.000,C 90.000,E1 260.849} C_DIS
LIN {X -0.077,Y -535.605,Z 956.243,A 0.000,B 0.000,C 90.000,E1 259.690} C_DIS
LIN {X -0.176,Y -532.729,Z 956.230,A 0.000,B 0.000,C 90.000,E1 257.409} C_DIS
LIN {X -0.114,Y -529.964,Z 956.217,A 0.000,B 0.000,C 90.000,E1 255.102} C_DIS
LIN {X -0.176,Y -528.000,Z 956.208,A 0.000,B 0.000,C 90.000,E1 253.378} C_DIS
LIN {X 0.191,Y -526.697,Z 956.201,A 0.000,B 0.000,C 90.000,E1 252.181} C_DIS
LIN {X -0.130,Y -524.538,Z 956.192,A 0.000,B 0.000,C 90.000,E1 250.477} C_DIS
LIN {X -0.166,Y -522.683,Z 956.183,A 0.000,B 0.000,C 90.000,E1 249.028} C_DIS
LIN {X 0.283,Y -520.392,Z 956.174,A 0.000,B 0.000,C 90.000,E1 247.230} C_DIS
LIN {X -0.080,Y -518.698,Z 956.167,A 0.000,B 0.000,C 90.000,E1 246.102} C_DIS
LIN {X 0.018,Y -515.959,Z 956.157,A 0.000,B 0.000,C 90.000,E1 244.332} C_DIS
LIN {X -0.068,Y -513.661,Z 956.149,A 0.000,B 0.000,C 90.000,E1 242.871} C_DIS
LIN {X -0.077,Y -510.794,Z 956.139,A 0.000,B 0.000,C 90.000,E1 241.101} C_DIS
LIN {X -0.007,Y -509.293,Z 956.135,A 0.000,B 0.000,C 90.000,E1 240.205} C_DIS
LIN {X -0.190,Y -506.519,Z 956.126,A 0.000,B 0.000,C 90.000,E1 238.742} C_DIS
LIN {X -0.043,Y -504.072,Z 956.120,A 0.000,B 0.000,C 90.000,E1 237.533} C_DIS
LIN {X -0.082,Y -501.453,Z 956.113,A 0.000,B 0.000,C 90.000,E1 236.342} C_DIS
LIN {X 0.007,Y -497.307,Z 956.103,A 0.000,B 0.000,C 90.000,E1 234.529} C_DIS
LIN {X -0.008,Y -493.293,Z 956.093,A 0.000,B 0.000,C 90.000,E1 232.718} C_DIS
LIN {X 0.079,Y -489.154,Z 956.083,A 0.000,B 0.000,C 90.000,E1 230.884} C_DIS
LIN {X -0.127,Y -485.620,Z 956.074,A 0.000,B 0.000,C 90.000,E1 229.380} C_DIS
LIN {X -0.267,Y -481.411,Z 956.064,A 0.000,B 0.000,C 90.000,E1 227.553} C_DIS
LIN {X -0.092,Y -478.604,Z 956.057,A 0.000,B 0.000,C 90.000,E1 226.296} C_DIS
LIN {X 0.036,Y -475.890,Z 956.050,A 0.000,B 0.000,C 90.000,E1 225.040} C_DIS
LIN {X -0.013,Y -471.743,Z 956.040,A 0.000,B 0.000,C 90.000,E1 223.176} C_DIS
LIN {X -0.073,Y -467.009,Z 956.028,A 0.000,B 0.000,C 90.000,E1 220.987} C_DIS
LIN {X -0.026,Y -463.464,Z 956.019,A 0.000,B 0.000,C 90.000,E1 219.402} C_DIS
LIN {X 0.020,Y -459.994,Z 956.010,A 0.000,B 0.000,C 90.000,E1 217.810} C_DIS
LIN {X -0.111,Y -457.858,Z 956.005,A 0.000,B 0.000,C 90.000,E1 216.870} C_DIS
LIN {X 0.191,Y -454.290,Z 955.996,A 0.000,B 0.000,C 90.000,E1 215.231} C_DIS
LIN {X 0.240,Y -450.083,Z 955.985,A 0.000,B 0.000,C 90.000,E1 213.293} C_DIS
LIN {X -0.056,Y -445.835,Z 955.974,A 0.000,B 0.000,C 90.000,E1 211.386} C_DIS
LIN {X 0.030,Y -442.275,Z 955.965,A 0.000,B 0.000,C 90.000,E1 209.745} C_DIS
LIN {X 0.052,Y -438.726,Z 955.956,A 0.000,B 0.000,C 90.000,E1 208.103} C_DIS
LIN {X -0.203,Y -435.128,Z 955.947,A 0.000,B 0.000,C 90.000,E1 206.488} C_DIS
LIN {X -0.145,Y -432.193,Z 955.940,A 0.000,B 0.000,C 90.000,E1 205.155} C_DIS
LIN {X 0.053,Y -429.958,Z 955.934,A 0.000,B 0.000,C 90.000,E1 204.131} C_DIS
LIN {X -0.157,Y -425.373,Z 955.923,A 0.000,B 0.000,C 90.000,E1 202.153} C_DIS
LIN {X -0.119,Y -419.583,Z 955.908,A 0.000,B 0.000,C 90.000,E1 199.450} C_DIS
LIN {X 0.090,Y -414.716,Z 955.895,A 0.000,B 0.000,C 90.000,E1 197.040} C_DIS
LIN {X 0.150,Y -412.032,Z 955.887,A 0.000,B 0.000,C 90.000,E1 195.662} C_DIS
LIN {X 0.054,Y -409.278,Z 955.880,A 0.000,B 0.000,C 90.000,E1 194.300} C_DIS
LIN {X -0.075,Y -405.837,Z 955.870,A 0.000,B 0.000,C 90.000,E1 192.591} C_DIS
LIN {X 0.038,Y -402.502,Z 955.860,A 0.000,B 0.000,C 90.000,E1 190.838} C_DIS
LIN {X 0.022,Y -399.886,Z 955.853,A 0.000,B 0.000,C 90.000,E1 189.443} C_DIS
LIN {X -0.059,Y -396.508,Z 955.843,A 0.000,B 0.000,C 90.000,E1 187.701} C_DIS
LIN {X 0.041,Y -392.583,Z 955.831,A 0.000,B 0.000,C 90.000,E1 185.568} C_DIS
LIN {X 0.143,Y -387.616,Z 955.813,A 0.000,B 0.000,C 90.000,E1 182.350} C_DIS
LIN {X -0.130,Y -386.723,Z 955.807,A 0.000,B 0.000,C 90.000,E1 181.318} C_DIS
LIN {X 0.059,Y -386.584,Z 955.803,A 0.000,B 0.000,C 90.000,E1 180.573} C_DIS
LIN {X -0.089,Y -386.789,Z 955.800,A 0.000,B 0.000,C 90.000,E1 180.057} C_DIS
LIN {X -0.128,Y -387.851,Z 955.796,A 0.000,B 0.000,C 90.000,E1 179.312} C_DIS
LIN {X 0.123,Y -388.964,Z 955.793,A 0.000,B 0.000,C 90.000,E1 178.740} C_DIS
LIN {X -0.010,Y -391.104,Z 955.790,A 0.000,B 0.000,C 90.000,E1 178.224} C_DIS
LIN {X -0.095,Y -394.184,Z 955.787,A 0.000,B 0.000,C 90.000,E1 177.707} C_DIS
LIN {X -0.106,Y -395.383,Z 955.786,A 0.000,B 0.000,C 90.000,E1 177.535} C_DIS
LIN {X -0.122,Y -398.753,Z 955.784,A 0.000,B 0.000,C 90.000,E1 177.135} C_DIS
LIN {X -0.023,Y -406.170,Z 955.780,A 0.000,B 0.000,C 90.000,E1 176.388} C_DIS
LIN {X -0.081,Y -418.123,Z 955.774,A 0.000,B 0.000,C 90.000,E1 175.355} C_DIS
LIN {X 0.071,Y -430.583,Z 955.768,A 0.000,B 0.000,C 90.000,E1 174.261} C_DIS
LIN {X -0.091,Y -434.762,Z 955.766,A 0.000,B 0.000,C 90.000,E1 173.913} C_DIS
LIN {X -0.006,Y -442.219,Z 955.762,A 0.000,B 0.000,C 90.000,E1 173.223} C_DIS
LIN {X -0.006,Y -452.506,Z 955.757,A 0.000,B 0.000,C 90.000,E1 172.243} C_DIS
LIN {X 0.061,Y -459.418,Z 955.753,A 0.000,B 0.000,C 90.000,E1 171.546} C_DIS
LIN {X 0.216,Y -470.150,Z 955.747,A 0.000,B 0.000,C 90.000,E1 170.387} C_DIS
LIN {X 0.106,Y -475.429,Z 955.743,A 0.000,B 0.000,C 90.000,E1 169.803} C_DIS
LIN {X -0.145,Y -484.519,Z 955.737,A 0.000,B 0.000,C 90.000,E1 168.757} C_DIS
LIN {X 0.114,Y -491.726,Z 955.732,A 0.000,B 0.000,C 90.000,E1 167.825} C_DIS
LIN {X 0.096,Y -501.920,Z 955.725,A 0.000,B 0.000,C 90.000,E1 166.464} C_DIS
LIN {X 0.131,Y -511.362,Z 955.717,A 0.000,B 0.000,C 90.000,E1 165.117} C_DIS
LIN {X 0.296,Y -517.070,Z 955.713,A 0.000,B 0.000,C 90.000,E1 164.212} C_DIS
LIN {X -0.244,Y -520.939,Z 955.709,A 0.000,B 0.000,C 90.000,E1 163.685} C_DIS
LIN {X -0.135,Y -527.304,Z 955.704,A 0.000,B 0.000,C 90.000,E1 162.653} C_DIS
LIN {X 0.254,Y -534.448,Z 955.697,A 0.000,B 0.000,C 90.000,E1 161.456} C_DIS
LIN {X -0.276,Y -541.436,Z 955.691,A 0.000,B 0.000,C 90.000,E1 160.369} C_DIS
LIN {X -0.020,Y -548.228,Z 955.685,A 0.000,B 0.000,C 90.000,E1 159.209} C_DIS
LIN {X -0.177,Y -554.810,Z 955.678,A 0.000,B 0.000,C 90.000,E1 158.103} C_DIS
LIN {X -0.030,Y -561.068,Z 955.672,A 0.000,B 0.000,C 90.000,E1 156.975} C_DIS
LIN {X -0.242,Y -564.786,Z 955.668,A 0.000,B 0.000,C 90.000,E1 156.305} C_DIS
LIN {X -0.042,Y -571.110,Z 955.661,A 0.000,B 0.000,C 90.000,E1 155.049} C_DIS
LIN {X 0.056,Y -574.421,Z 955.658,A 0.000,B 0.000,C 90.000,E1 154.357} C_DIS
LIN {X 0.002,Y -581.033,Z 955.649,A 0.000,B 0.000,C 90.000,E1 152.871} C_DIS
LIN {X -0.131,Y -584.389,Z 955.645,A 0.000,B 0.000,C 90.000,E1 152.076} C_DIS
LIN {X -0.111,Y -588.520,Z 955.639,A 0.000,B 0.000,C 90.000,E1 151.001} C_DIS
LIN {X -0.054,Y -590.524,Z 955.636,A 0.000,B 0.000,C 90.000,E1 150.461} C_DIS
LIN {X -0.185,Y -597.084,Z 955.626,A 0.000,B 0.000,C 90.000,E1 148.614} C_DIS
LIN {X 0.164,Y -599.747,Z 955.621,A 0.000,B 0.000,C 90.000,E1 147.788} C_DIS
LIN {X 0.047,Y -605.812,Z 955.611,A 0.000,B 0.000,C 90.000,E1 145.960} C_DIS
LIN {X -0.306,Y -610.201,Z 955.604,A 0.000,B 0.000,C 90.000,E1 144.689} C_DIS
LIN {X -0.289,Y -615.405,Z 955.595,A 0.000,B 0.000,C 90.000,E1 143.130} C_DIS
LIN {X 0.210,Y -620.549,Z 955.586,A 0.000,B 0.000,C 90.000,E1 141.537} C_DIS
LIN {X 0.329,Y -625.574,Z 955.578,A 0.000,B 0.000,C 90.000,E1 139.989} C_DIS
LIN {X 0.064,Y -630.659,Z 955.569,A 0.000,B 0.000,C 90.000,E1 138.485} C_DIS
LIN {X 0.213,Y -636.941,Z 955.560,A 0.000,B 0.000,C 90.000,E1 136.701} C_DIS
LIN {X -0.249,Y -641.392,Z 955.553,A 0.000,B 0.000,C 90.000,E1 135.486} C_DIS
LIN {X 0.138,Y -647.666,Z 955.543,A 0.000,B 0.000,C 90.000,E1 133.704} C_DIS
LIN {X 0.372,Y -651.287,Z 955.537,A 0.000,B 0.000,C 90.000,E1 132.690} C_DIS
LIN {X 0.054,Y -658.622,Z 955.526,A 0.000,B 0.000,C 90.000,E1 130.744} C_DIS
LIN {X 0.053,Y -663.270,Z 955.520,A 0.000,B 0.000,C 90.000,E1 129.519} C_DIS
LIN {X -0.393,Y -668.765,Z 955.512,A 0.000,B 0.000,C 90.000,E1 128.096} C_DIS
LIN {X 0.202,Y -672.278,Z 955.506,A 0.000,B 0.000,C 90.000,E1 127.076} C_DIS
LIN {X 0.037,Y -676.474,Z 955.499,A 0.000,B 0.000,C 90.000,E1 125.884} C_DIS
LIN {X -0.214,Y -678.836,Z 955.495,A 0.000,B 0.000,C 90.000,E1 125.185} C_DIS
LIN {X -0.271,Y -682.561,Z 955.489,A 0.000,B 0.000,C 90.000,E1 123.992} C_DIS
LIN {X 0.294,Y -685.885,Z 955.482,A 0.000,B 0.000,C 90.000,E1 122.752} C_DIS
LIN {X -0.247,Y -687.750,Z 955.478,A 0.000,B 0.000,C 90.000,E1 122.084} C_DIS
LIN {X -0.188,Y -690.127,Z 955.473,A 0.000,B 0.000,C 90.000,E1 121.131} C_DIS
LIN {X -0.096,Y -691.675,Z 955.469,A 0.000,B 0.000,C 90.000,E1 120.413} C_DIS
LIN {X 0.362,Y -693.074,Z 955.465,A 0.000,B 0.000,C 90.000,E1 119.667} C_DIS
LIN {X -0.119,Y -694.283,Z 955.461,A 0.000,B 0.000,C 90.000,E1 118.999} C_DIS
LIN {X 0.266,Y -695.571,Z 955.456,A 0.000,B 0.000,C 90.000,E1 118.025} C_DIS
LIN {X 0.093,Y -696.343,Z 955.452,A 0.000,B 0.000,C 90.000,E1 117.334} C_DIS
LIN {X 0.143,Y -697.147,Z 955.445,A 0.000,B 0.000,C 90.000,E1 116.155} C_DIS
LIN {X -0.414,Y -697.566,Z 955.439,A 0.000,B 0.000,C 90.000,E1 115.027} C_DIS
LIN {X 0.081,Y -697.687,Z 955.435,A 0.000,B 0.000,C 90.000,E1 114.283} C_DIS
LIN {X -0.035,Y -697.437,Z 955.432,A 0.000,B 0.000,C 90.000,E1 113.823} C_DIS
LIN {X -0.056,Y -697.040,Z 955.431,A 0.000,B 0.000,C 90.000,E1 113.590} C_DIS
LIN {X -0.183,Y -695.717,Z 955.428,A 0.000,B 0.000,C 90.000,E1 113.131} C_DIS
LIN {X -0.203,Y -694.459,Z 955.427,A 0.000,B 0.000,C 90.000,E1 112.898} C_DIS
LIN {X 0.165,Y -692.168,Z 955.425,A 0.000,B 0.000,C 90.000,E1 112.514} C_DIS
LIN {X 0.021,Y -691.234,Z 955.425,A 0.000,B 0.000,C 90.000,E1 112.408} C_DIS
LIN {X 0.139,Y -689.837,Z 955.424,A 0.000,B 0.000,C 90.000,E1 112.280} C_DIS
LIN {X -0.239,Y -684.489,Z 955.422,A 0.000,B 0.000,C 90.000,E1 112.025} C_DIS
LIN {X -0.022,Y -680.741,Z 955.421,A 0.000,B 0.000,C 90.000,E1 111.844} C_DIS
LIN {X -0.157,Y -676.035,Z 955.421,A 0.000,B 0.000,C 90.000,E1 111.716} C_DIS
LIN {X 0.212,Y -674.535,Z 955.420,A 0.000,B 0.000,C 90.000,E1 111.663} C_DIS
LIN {X -0.148,Y -667.396,Z 955.420,A 0.000,B 0.000,C 90.000,E1 111.642} C_DIS
LIN {X -0.180,Y -631.281,Z 955.420,A 0.000,B 0.000,C 90.000,E1 111.642} C_DIS
LIN {X 0.246,Y -626.326,Z 955.420,A 0.000,B 0.000,C 90.000,E1 111.535} C_DIS
LIN {X -0.150,Y -620.711,Z 955.419,A 0.000,B 0.000,C 90.000,E1 111.461} C_DIS
LIN {X 0.168,Y -615.101,Z 955.418,A 0.000,B 0.000,C 90.000,E1 111.280} C_DIS
LIN {X 0.090,Y -609.713,Z 955.417,A 0.000,B 0.000,C 90.000,E1 111.099} C_DIS
LIN {X 0.182,Y -606.677,Z 955.417,A 0.000,B 0.000,C 90.000,E1 110.972} C_DIS
LIN {X -0.013,Y -600.082,Z 955.415,A 0.000,B 0.000,C 90.000,E1 110.663} C_DIS
LIN {X 0.142,Y -593.537,Z 955.413,A 0.000,B 0.000,C 90.000,E1 110.248} C_DIS
LIN {X 0.060,Y -576.927,Z 955.406,A 0.000,B 0.000,C 90.000,E1 109.033} C_DIS
LIN {X -0.141,Y -573.228,Z 955.405,A 0.000,B 0.000,C 90.000,E1 108.833} C_DIS
LIN {X -0.187,Y -566.970,Z 955.403,A 0.000,B 0.000,C 90.000,E1 108.489} C_DIS
LIN {X -0.039,Y -556.761,Z 955.400,A 0.000,B 0.000,C 90.000,E1 108.000} C_DIS
LIN {X -0.150,Y -553.085,Z 955.399,A 0.000,B 0.000,C 90.000,E1 107.819} C_DIS
LIN {X 0.154,Y -551.544,Z 955.398,A 0.000,B 0.000,C 90.000,E1 107.638} C_DIS
LIN {X 0.115,Y -551.526,Z 955.398,A 0.000,B 0.000,C 90.000,E1 107.638} C_DIS
LIN {X 0.160,Y -550.949,Z 955.397,A 0.000,B 0.000,C 90.000,E1 107.402} C_DIS
LIN {X -0.102,Y -550.799,Z 955.395,A 0.000,B 0.000,C 90.000,E1 107.149} C_DIS
LIN {X 0.232,Y -551.634,Z 955.381,A 0.000,B 0.000,C 90.000,E1 104.592} C_DIS
LIN {X -0.087,Y -553.308,Z 955.366,A 0.000,B 0.000,C 90.000,E1 101.827} C_DIS
LIN {X 0.268,Y -555.245,Z 955.353,A 0.000,B 0.000,C 90.000,E1 99.557} C_DIS
LIN {X -0.221,Y -556.743,Z 955.344,A 0.000,B 0.000,C 90.000,E1 97.936} C_DIS
LIN {X 0.230,Y -557.727,Z 955.338,A 0.000,B 0.000,C 90.000,E1 96.777} C_DIS
LIN {X 0.072,Y -558.548,Z 955.332,A 0.000,B 0.000,C 90.000,E1 95.682} C_DIS
LIN {X 0.004,Y -559.456,Z 955.324,A 0.000,B 0.000,C 90.000,E1 94.302} C_DIS
LIN {X 0.035,Y -560.415,Z 955.315,A 0.000,B 0.000,C 90.000,E1 92.636} C_DIS
LIN {X -0.040,Y -561.103,Z 955.307,A 0.000,B 0.000,C 90.000,E1 91.260} C_DIS
LIN {X -0.116,Y -561.655,Z 955.299,A 0.000,B 0.000,C 90.000,E1 89.885} C_DIS
LIN {X -0.084,Y -562.095,Z 955.290,A 0.000,B 0.000,C 90.000,E1 88.224} C_DIS
LIN {X -0.106,Y -562.428,Z 955.282,A 0.000,B 0.000,C 90.000,E1 86.846} C_DIS
LIN {X -0.146,Y -562.666,Z 955.275,A 0.000,B 0.000,C 90.000,E1 85.469} C_DIS
LIN {X -0.003,Y -562.875,Z 955.266,A 0.000,B 0.000,C 90.000,E1 83.799} C_DIS
LIN {X 0.140,Y -563.170,Z 955.256,A 0.000,B 0.000,C 90.000,E1 82.129} C_DIS
LIN {X -0.112,Y -563.582,Z 955.247,A 0.000,B 0.000,C 90.000,E1 80.500} C_DIS
LIN {X -0.178,Y -564.408,Z 955.237,A 0.000,B 0.000,C 90.000,E1 78.578} C_DIS
LIN {X 0.048,Y -565.581,Z 955.224,A 0.000,B 0.000,C 90.000,E1 76.353} C_DIS
LIN {X -0.077,Y -566.476,Z 955.217,A 0.000,B 0.000,C 90.000,E1 74.991} C_DIS
LIN {X -0.247,Y -567.768,Z 955.206,A 0.000,B 0.000,C 90.000,E1 73.087} C_DIS
LIN {X -0.007,Y -568.608,Z 955.198,A 0.000,B 0.000,C 90.000,E1 71.692} C_DIS
LIN {X -0.085,Y -569.227,Z 955.192,A 0.000,B 0.000,C 90.000,E1 70.604} C_DIS
LIN {X -0.162,Y -569.692,Z 955.186,A 0.000,B 0.000,C 90.000,E1 69.518} C_DIS
LIN {X -0.217,Y -570.231,Z 955.179,A 0.000,B 0.000,C 90.000,E1 68.156} C_DIS
LIN {X 0.091,Y -570.682,Z 955.169,A 0.000,B 0.000,C 90.000,E1 66.485} C_DIS
LIN {X 0.114,Y -571.097,Z 955.160,A 0.000,B 0.000,C 90.000,E1 64.845} C_DIS
LIN {X 0.138,Y -571.400,Z 955.151,A 0.000,B 0.000,C 90.000,E1 63.204} C_DIS
LIN {X 0.073,Y -571.543,Z 955.144,A 0.000,B 0.000,C 90.000,E1 61.847} C_DIS
LIN {X 0.117,Y -571.617,Z 955.135,A 0.000,B 0.000,C 90.000,E1 60.205} C_DIS
LIN {X -0.211,Y -571.829,Z 955.124,A 0.000,B 0.000,C 90.000,E1 58.329} C_DIS
LIN {X -0.178,Y -571.779,Z 955.116,A 0.000,B 0.000,C 90.000,E1 56.962} C_DIS
LIN {X -0.148,Y -571.433,Z 955.109,A 0.000,B 0.000,C 90.000,E1 55.595} C_DIS
LIN {X 0.195,Y -570.998,Z 955.101,A 0.000,B 0.000,C 90.000,E1 54.196} C_DIS
LIN {X -0.068,Y -570.493,Z 955.095,A 0.000,B 0.000,C 90.000,E1 53.130} C_DIS
LIN {X 0.008,Y -569.655,Z 955.089,A 0.000,B 0.000,C 90.000,E1 52.029} C_DIS
LIN {X 0.077,Y -568.668,Z 955.083,A 0.000,B 0.000,C 90.000,E1 50.928} C_DIS
LIN {X 0.129,Y -567.494,Z 955.077,A 0.000,B 0.000,C 90.000,E1 49.828} C_DIS
LIN {X 0.043,Y -566.449,Z 955.072,A 0.000,B 0.000,C 90.000,E1 49.013} C_DIS
LIN {X 0.316,Y -565.155,Z 955.068,A 0.000,B 0.000,C 90.000,E1 48.162} C_DIS
LIN {X 0.256,Y -563.130,Z 955.062,A 0.000,B 0.000,C 90.000,E1 47.067} C_DIS
LIN {X 0.166,Y -560.857,Z 955.056,A 0.000,B 0.000,C 90.000,E1 45.972} C_DIS
LIN {X -0.026,Y -558.795,Z 955.051,A 0.000,B 0.000,C 90.000,E1 45.162} C_DIS
LIN {X -0.238,Y -556.431,Z 955.046,A 0.000,B 0.000,C 90.000,E1 44.352} C_DIS
LIN {X -0.074,Y -553.824,Z 955.042,A 0.000,B 0.000,C 90.000,E1 43.500} C_DIS
LIN {X 0.015,Y -551.922,Z 955.039,A 0.000,B 0.000,C 90.000,E1 42.933} C_DIS
LIN {X 0.131,Y -548.797,Z 955.034,A 0.000,B 0.000,C 90.000,E1 42.081} C_DIS
LIN {X -0.029,Y -547.107,Z 955.032,A 0.000,B 0.000,C 90.000,E1 41.676} C_DIS
LIN {X 0.153,Y -542.107,Z 955.025,A 0.000,B 0.000,C 90.000,E1 40.539} C_DIS
LIN {X -0.197,Y -537.717,Z 955.021,A 0.000,B 0.000,C 90.000,E1 39.725} C_DIS
LIN {X 0.160,Y -533.069,Z 955.016,A 0.000,B 0.000,C 90.000,E1 38.830} C_DIS
LIN {X 0.111,Y -526.264,Z 955.009,A 0.000,B 0.000,C 90.000,E1 37.684} C_DIS
LIN {X 0.150,Y -519.961,Z 955.004,A 0.000,B 0.000,C 90.000,E1 36.664} C_DIS
LIN {X 0.045,Y -516.151,Z 955.001,A 0.000,B 0.000,C 90.000,E1 36.091} C_DIS
LIN {X -0.165,Y -510.149,Z 954.996,A 0.000,B 0.000,C 90.000,E1 35.231} C_DIS
LIN {X -0.119,Y -504.680,Z 954.992,A 0.000,B 0.000,C 90.000,E1 34.485} C_DIS
LIN {X -0.223,Y -502.421,Z 954.990,A 0.000,B 0.000,C 90.000,E1 34.199} C_DIS
LIN {X 0.308,Y -493.646,Z 954.984,A 0.000,B 0.000,C 90.000,E1 33.086} C_DIS
LIN {X -0.184,Y -488.244,Z 954.981,A 0.000,B 0.000,C 90.000,E1 32.546} C_DIS
LIN {X 0.186,Y -482.597,Z 954.978,A 0.000,B 0.000,C 90.000,E1 31.926} C_DIS
LIN {X -0.031,Y -474.199,Z 954.973,A 0.000,B 0.000,C 90.000,E1 31.131} C_DIS
LIN {X -0.164,Y -466.781,Z 954.969,A 0.000,B 0.000,C 90.000,E1 30.463} C_DIS
LIN {X -0.149,Y -456.583,Z 954.964,A 0.000,B 0.000,C 90.000,E1 29.539} C_DIS
LIN {X -0.030,Y -444.433,Z 954.958,A 0.000,B 0.000,C 90.000,E1 28.487} C_DIS
LIN {X -0.072,Y -424.724,Z 954.949,A 0.000,B 0.000,C 90.000,E1 26.796} C_DIS
LIN {X 0.177,Y -408.328,Z 954.940,A 0.000,B 0.000,C 90.000,E1 25.207} C_DIS
LIN {X -0.044,Y -399.559,Z 954.935,A 0.000,B 0.000,C 90.000,E1 24.335} C_DIS
LIN {X 0.080,Y -396.016,Z 954.933,A 0.000,B 0.000,C 90.000,E1 23.898} C_DIS
LIN {X 0.158,Y -393.531,Z 954.931,A 0.000,B 0.000,C 90.000,E1 23.515} C_DIS
LIN {X -0.177,Y -392.441,Z 954.930,A 0.000,B 0.000,C 90.000,E1 23.387} C_DIS
LIN {X -0.091,Y -390.827,Z 954.928,A 0.000,B 0.000,C 90.000,E1 23.003} C_DIS
LIN {X 0.023,Y -390.482,Z 954.927,A 0.000,B 0.000,C 90.000,E1 22.898} C_DIS
LIN {X -0.051,Y -390.139,Z 954.926,A 0.000,B 0.000,C 90.000,E1 22.642} C_DIS
LIN {X -0.014,Y -389.512,Z 954.924,A 0.000,B 0.000,C 90.000,E1 22.280} C_DIS
LIN {X -0.158,Y -389.454,Z 954.920,A 0.000,B 0.000,C 90.000,E1 21.589} C_DIS
LIN {X 0.170,Y -390.570,Z 954.910,A 0.000,B 0.000,C 90.000,E1 19.758} C_DIS
LIN {X -0.152,Y -394.679,Z 954.888,A 0.000,B 0.000,C 90.000,E1 15.898} C_DIS
LIN {X -0.072,Y -398.289,Z 954.873,A 0.000,B 0.000,C 90.000,E1 13.063} C_DIS
LIN {X -0.048,Y -403.051,Z 954.855,A 0.000,B 0.000,C 90.000,E1 9.905} C_DIS
LIN {X -0.025,Y -407.264,Z 954.841,A 0.000,B 0.000,C 90.000,E1 7.466} C_DIS
LIN {X -0.015,Y -412.564,Z 954.826,A 0.000,B 0.000,C 90.000,E1 4.702} C_DIS
LIN {X 0.069,Y -417.656,Z 954.813,A 0.000,B 0.000,C 90.000,E1 2.293} C_DIS
LIN {X 0.207,Y -424.533,Z 954.797,A 0.000,B 0.000,C 90.000,E1 359.427} C_DIS
LIN {X -0.170,Y -425.765,Z 954.795,A 0.000,B 0.000,C 90.000,E1 359.141} C_DIS
LIN {X -0.179,Y -428.458,Z 954.792,A 0.000,B 0.000,C 90.000,E1 358.568} C_DIS
LIN {X -0.147,Y -429.491,Z 954.791,A 0.000,B 0.000,C 90.000,E1 358.396} C_DIS
LIN {X -0.116,Y -430.802,Z 954.790,A 0.000,B 0.000,C 90.000,E1 358.224} C_DIS
LIN {X -0.169,Y -434.168,Z 954.788,A 0.000,B 0.000,C 90.000,E1 357.879} C_DIS
LIN {X -0.017,Y -436.167,Z 954.787,A 0.000,B 0.000,C 90.000,E1 357.707} C_DIS
LIN {X -0.214,Y -440.207,Z 954.786,A 0.000,B 0.000,C 90.000,E1 357.478} C_DIS
LIN {X 0.213,Y -454.828,Z 954.782,A 0.000,B 0.000,C 90.000,E1 356.674} C_DIS
LIN {X 0.025,Y -465.078,Z 954.779,A 0.000,B 0.000,C 90.000,E1 356.159} C_DIS
LIN {X -0.092,Y -478.306,Z 954.775,A 0.000,B 0.000,C 90.000,E1 355.469} C_DIS
LIN {X -0.033,Y -492.789,Z 954.770,A 0.000,B 0.000,C 90.000,E1 354.666} C_DIS
LIN {X 0.133,Y -502.575,Z 954.767,A 0.000,B 0.000,C 90.000,E1 354.090} C_DIS
LIN {X -0.027,Y -510.730,Z 954.765,A 0.000,B 0.000,C 90.000,E1 353.628} C_DIS
LIN {X -0.148,Y -521.584,Z 954.761,A 0.000,B 0.000,C 90.000,E1 352.932} C_DIS
LIN {X 0.211,Y -527.700,Z 954.758,A 0.000,B 0.000,C 90.000,E1 352.470} C_DIS
LIN {X -0.159,Y -536.566,Z 954.755,A 0.000,B 0.000,C 90.000,E1 351.837} C_DIS
LIN {X -0.291,Y -542.214,Z 954.752,A 0.000,B 0.000,C 90.000,E1 351.376} C_DIS
LIN {X -0.156,Y -549.096,Z 954.748,A 0.000,B 0.000,C 90.000,E1 350.735} C_DIS
LIN {X 0.230,Y -555.488,Z 954.745,A 0.000,B 0.000,C 90.000,E1 350.038} C_DIS
